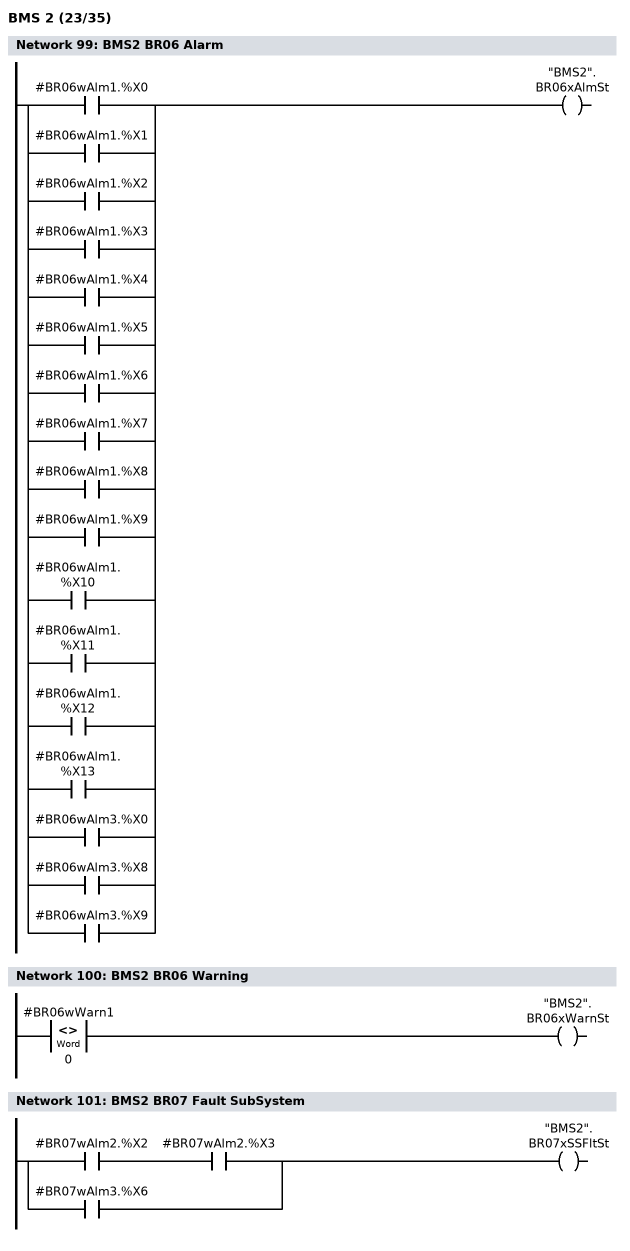
   RUNG wire#powerrail
      Contact( #BR06wAlm1.%X0 )
      wire#w1
      Coil( "BMS2".BR06xAlmSt )
   END_RUNG
   RUNG wire#powerrail
      Contact( #BR06wAlm1.%X1 )
   END_RUNG wire#w1
   RUNG wire#powerrail
      Contact( #BR06wAlm1.%X2 )
   END_RUNG wire#w1
   RUNG wire#powerrail
      Contact( #BR06wAlm1.%X3 )
   END_RUNG wire#w1
   RUNG wire#powerrail
      Contact( #BR06wAlm1.%X4 )
   END_RUNG wire#w1
   RUNG wire#powerrail
      Contact( #BR06wAlm1.%X5 )
   END_RUNG wire#w1
   RUNG wire#powerrail
      Contact( #BR06wAlm1.%X6 )
   END_RUNG wire#w1
   RUNG wire#powerrail
      Contact( #BR06wAlm1.%X7 )
   END_RUNG wire#w1
   RUNG wire#powerrail
      Contact( #BR06wAlm1.%X8 )
   END_RUNG wire#w1
   RUNG wire#powerrail
      Contact( #BR06wAlm1.%X9 )
   END_RUNG wire#w1
   RUNG wire#powerrail
      Contact( #BR06wAlm1.%X10 )
   END_RUNG wire#w1
   RUNG wire#powerrail
      Contact( #BR06wAlm1.%X11 )
   END_RUNG wire#w1
   RUNG wire#powerrail
      Contact( #BR06wAlm1.%X12 )
   END_RUNG wire#w1
   RUNG wire#powerrail
      Contact( #BR06wAlm1.%X13 )
   END_RUNG wire#w1
   RUNG wire#powerrail
      Contact( #BR06wAlm3.%X0 )
   END_RUNG wire#w1
   RUNG wire#powerrail
      Contact( #BR06wAlm3.%X8 )
   END_RUNG wire#w1
   RUNG wire#powerrail
      Contact( #BR06wAlm3.%X9 )
   END_RUNG wire#w1
   // the same network as SCL:
   "BMS2".BR06xAlmSt := #BR06wAlm1.%X0 OR #BR06wAlm1.%X1 OR #BR06wAlm1.%X2 OR #BR06wAlm1.%X3 OR #BR06wAlm1.%X4 OR #BR06wAlm1.%X5 OR #BR06wAlm1.%X6 OR #BR06wAlm1.%X7 OR #BR06wAlm1.%X8 OR #BR06wAlm1.%X9 OR #BR06wAlm1.%X10 OR #BR06wAlm1.%X11 OR #BR06wAlm1.%X12 OR #BR06wAlm1.%X13 OR #BR06wAlm3.%X0 OR #BR06wAlm3.%X8 OR #BR06wAlm3.%X9;
END_REGION

REGION Network 100: BMS2 BR06 Warning
   RUNG wire#powerrail
      { S7_Templates := "SrcType := Word" } NE_Contact(in1 := #BR06wWarn1, in2 := 0)
      Coil( "BMS2".BR06xWarnSt )
   END_RUNG
   // the same network as SCL:
   "BMS2".BR06xWarnSt := #BR06wWarn1 <> 0;
END_REGION

REGION Network 101: BMS2 BR07 Fault SubSystem
   RUNG wire#powerrail
      Contact( #BR07wAlm2.%X2 )
      Contact( #BR07wAlm2.%X3 )
      wire#w1
      Coil( "BMS2".BR07xSSFltSt )
   END_RUNG
   RUNG wire#powerrail
      Contact( #BR07wAlm3.%X6 )
   END_RUNG wire#w1
   // the same network as SCL:
   "BMS2".BR07xSSFltSt := (#BR07wAlm2.%X2 AND #BR07wAlm2.%X3) OR #BR07wAlm3.%X6;
END_REGION

REGION Network 102: BMS2 BR07 Fault
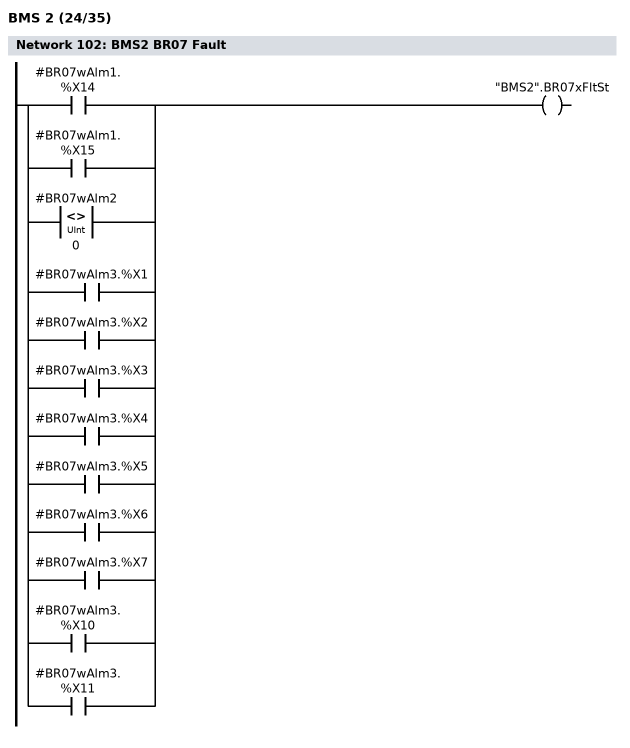
   RUNG wire#powerrail
      Contact( #BR07wAlm1.%X14 )
      wire#w1
      Coil( "BMS2".BR07xFltSt )
   END_RUNG
   RUNG wire#powerrail
      Contact( #BR07wAlm1.%X15 )
   END_RUNG wire#w1
   RUNG wire#powerrail
      { S7_Templates := "SrcType := UInt" } NE_Contact(in1 := #BR07wAlm2, in2 := 0)
   END_RUNG wire#w1
   RUNG wire#powerrail
      Contact( #BR07wAlm3.%X1 )
   END_RUNG wire#w1
   RUNG wire#powerrail
      Contact( #BR07wAlm3.%X2 )
   END_RUNG wire#w1
   RUNG wire#powerrail
      Contact( #BR07wAlm3.%X3 )
   END_RUNG wire#w1
   RUNG wire#powerrail
      Contact( #BR07wAlm3.%X4 )
   END_RUNG wire#w1
   RUNG wire#powerrail
      Contact( #BR07wAlm3.%X5 )
   END_RUNG wire#w1
   RUNG wire#powerrail
      Contact( #BR07wAlm3.%X6 )
   END_RUNG wire#w1
   RUNG wire#powerrail
      Contact( #BR07wAlm3.%X7 )
   END_RUNG wire#w1
   RUNG wire#powerrail
      Contact( #BR07wAlm3.%X10 )
   END_RUNG wire#w1
   RUNG wire#powerrail
      Contact( #BR07wAlm3.%X11 )
   END_RUNG wire#w1
   // the same network as SCL:
   "BMS2".BR07xFltSt := #BR07wAlm1.%X14 OR #BR07wAlm1.%X15 OR (#BR07wAlm2 <> 0) OR #BR07wAlm3.%X1 OR #BR07wAlm3.%X2 OR #BR07wAlm3.%X3 OR #BR07wAlm3.%X4 OR #BR07wAlm3.%X5 OR #BR07wAlm3.%X6 OR #BR07wAlm3.%X7 OR #BR07wAlm3.%X10 OR #BR07wAlm3.%X11;
END_REGION

REGION Network 103: BMS2 BR07 Alarm
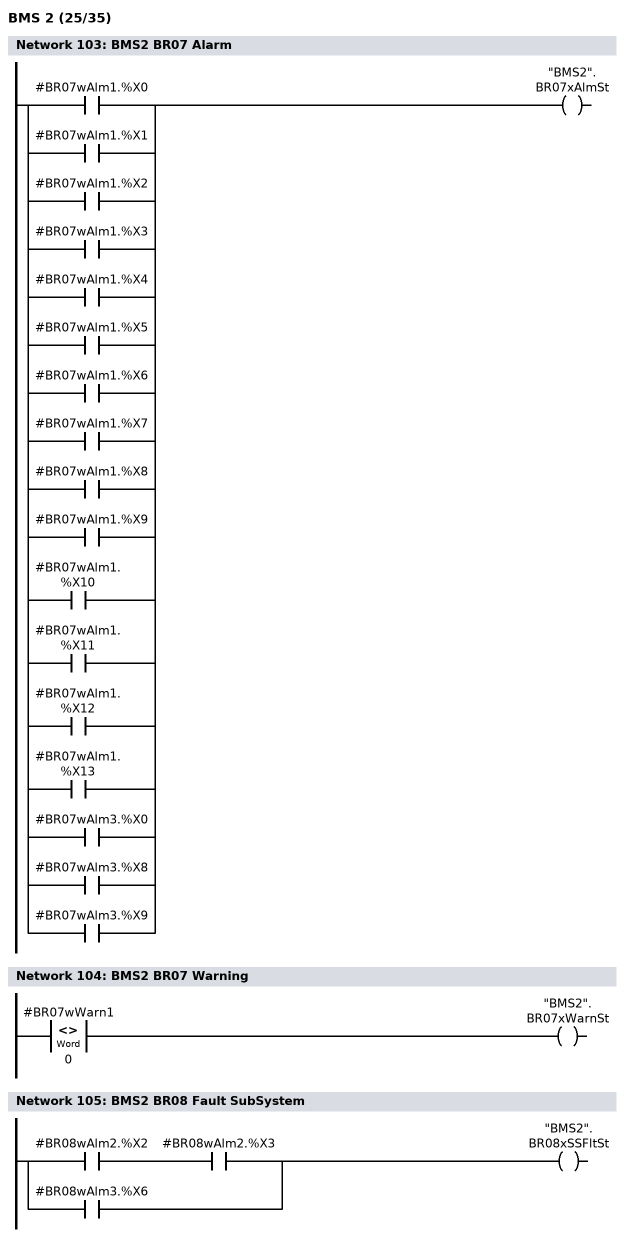
   RUNG wire#powerrail
      Contact( #BR07wAlm1.%X0 )
      wire#w1
      Coil( "BMS2".BR07xAlmSt )
   END_RUNG
   RUNG wire#powerrail
      Contact( #BR07wAlm1.%X1 )
   END_RUNG wire#w1
   RUNG wire#powerrail
      Contact( #BR07wAlm1.%X2 )
   END_RUNG wire#w1
   RUNG wire#powerrail
      Contact( #BR07wAlm1.%X3 )
   END_RUNG wire#w1
   RUNG wire#powerrail
      Contact( #BR07wAlm1.%X4 )
   END_RUNG wire#w1
   RUNG wire#powerrail
      Contact( #BR07wAlm1.%X5 )
   END_RUNG wire#w1
   RUNG wire#powerrail
      Contact( #BR07wAlm1.%X6 )
   END_RUNG wire#w1
   RUNG wire#powerrail
      Contact( #BR07wAlm1.%X7 )
   END_RUNG wire#w1
   RUNG wire#powerrail
      Contact( #BR07wAlm1.%X8 )
   END_RUNG wire#w1
   RUNG wire#powerrail
      Contact( #BR07wAlm1.%X9 )
   END_RUNG wire#w1
   RUNG wire#powerrail
      Contact( #BR07wAlm1.%X10 )
   END_RUNG wire#w1
   RUNG wire#powerrail
      Contact( #BR07wAlm1.%X11 )
   END_RUNG wire#w1
   RUNG wire#powerrail
      Contact( #BR07wAlm1.%X12 )
   END_RUNG wire#w1
   RUNG wire#powerrail
      Contact( #BR07wAlm1.%X13 )
   END_RUNG wire#w1
   RUNG wire#powerrail
      Contact( #BR07wAlm3.%X0 )
   END_RUNG wire#w1
   RUNG wire#powerrail
      Contact( #BR07wAlm3.%X8 )
   END_RUNG wire#w1
   RUNG wire#powerrail
      Contact( #BR07wAlm3.%X9 )
   END_RUNG wire#w1
   // the same network as SCL:
   "BMS2".BR07xAlmSt := #BR07wAlm1.%X0 OR #BR07wAlm1.%X1 OR #BR07wAlm1.%X2 OR #BR07wAlm1.%X3 OR #BR07wAlm1.%X4 OR #BR07wAlm1.%X5 OR #BR07wAlm1.%X6 OR #BR07wAlm1.%X7 OR #BR07wAlm1.%X8 OR #BR07wAlm1.%X9 OR #BR07wAlm1.%X10 OR #BR07wAlm1.%X11 OR #BR07wAlm1.%X12 OR #BR07wAlm1.%X13 OR #BR07wAlm3.%X0 OR #BR07wAlm3.%X8 OR #BR07wAlm3.%X9;
END_REGION

REGION Network 104: BMS2 BR07 Warning
   RUNG wire#powerrail
      { S7_Templates := "SrcType := Word" } NE_Contact(in1 := #BR07wWarn1, in2 := 0)
      Coil( "BMS2".BR07xWarnSt )
   END_RUNG
   // the same network as SCL:
   "BMS2".BR07xWarnSt := #BR07wWarn1 <> 0;
END_REGION

REGION Network 105: BMS2 BR08 Fault SubSystem
   RUNG wire#powerrail
      Contact( #BR08wAlm2.%X2 )
      Contact( #BR08wAlm2.%X3 )
      wire#w1
      Coil( "BMS2".BR08xSSFltSt )
   END_RUNG
   RUNG wire#powerrail
      Contact( #BR08wAlm3.%X6 )
   END_RUNG wire#w1
   // the same network as SCL:
   "BMS2".BR08xSSFltSt := (#BR08wAlm2.%X2 AND #BR08wAlm2.%X3) OR #BR08wAlm3.%X6;
END_REGION

REGION Network 106: BMS2 BR08 Fault
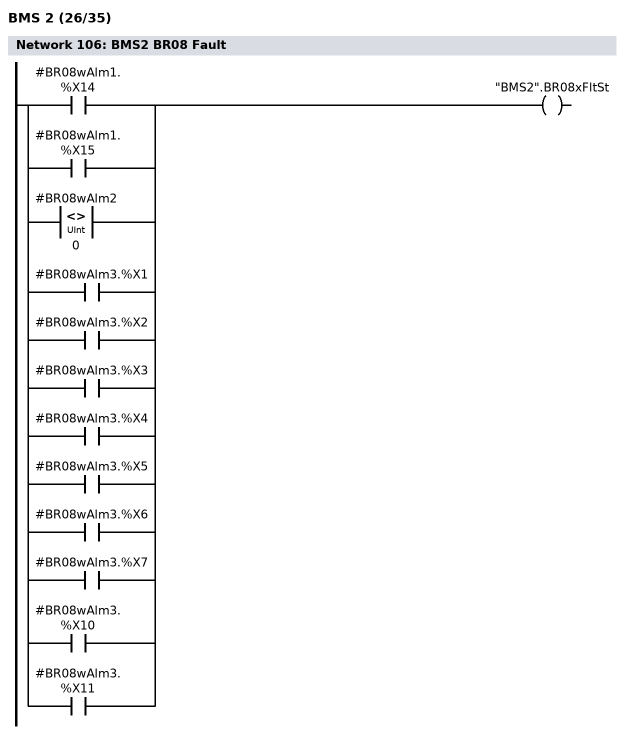
   RUNG wire#powerrail
      Contact( #BR08wAlm1.%X14 )
      wire#w1
      Coil( "BMS2".BR08xFltSt )
   END_RUNG
   RUNG wire#powerrail
      Contact( #BR08wAlm1.%X15 )
   END_RUNG wire#w1
   RUNG wire#powerrail
      { S7_Templates := "SrcType := UInt" } NE_Contact(in1 := #BR08wAlm2, in2 := 0)
   END_RUNG wire#w1
   RUNG wire#powerrail
      Contact( #BR08wAlm3.%X1 )
   END_RUNG wire#w1
   RUNG wire#powerrail
      Contact( #BR08wAlm3.%X2 )
   END_RUNG wire#w1
   RUNG wire#powerrail
      Contact( #BR08wAlm3.%X3 )
   END_RUNG wire#w1
   RUNG wire#powerrail
      Contact( #BR08wAlm3.%X4 )
   END_RUNG wire#w1
   RUNG wire#powerrail
      Contact( #BR08wAlm3.%X5 )
   END_RUNG wire#w1
   RUNG wire#powerrail
      Contact( #BR08wAlm3.%X6 )
   END_RUNG wire#w1
   RUNG wire#powerrail
      Contact( #BR08wAlm3.%X7 )
   END_RUNG wire#w1
   RUNG wire#powerrail
      Contact( #BR08wAlm3.%X10 )
   END_RUNG wire#w1
   RUNG wire#powerrail
      Contact( #BR08wAlm3.%X11 )
   END_RUNG wire#w1
   // the same network as SCL:
   "BMS2".BR08xFltSt := #BR08wAlm1.%X14 OR #BR08wAlm1.%X15 OR (#BR08wAlm2 <> 0) OR #BR08wAlm3.%X1 OR #BR08wAlm3.%X2 OR #BR08wAlm3.%X3 OR #BR08wAlm3.%X4 OR #BR08wAlm3.%X5 OR #BR08wAlm3.%X6 OR #BR08wAlm3.%X7 OR #BR08wAlm3.%X10 OR #BR08wAlm3.%X11;
END_REGION

REGION Network 107: BMS2 BR08 Alarm
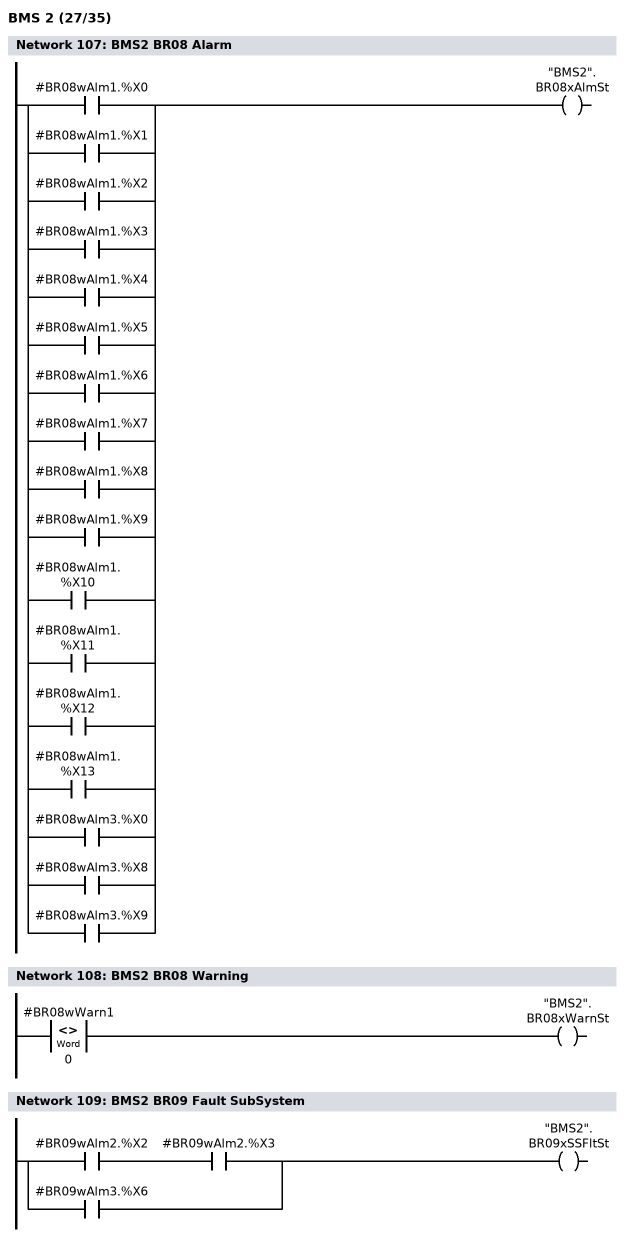
   RUNG wire#powerrail
      Contact( #BR08wAlm1.%X0 )
      wire#w1
      Coil( "BMS2".BR08xAlmSt )
   END_RUNG
   RUNG wire#powerrail
      Contact( #BR08wAlm1.%X1 )
   END_RUNG wire#w1
   RUNG wire#powerrail
      Contact( #BR08wAlm1.%X2 )
   END_RUNG wire#w1
   RUNG wire#powerrail
      Contact( #BR08wAlm1.%X3 )
   END_RUNG wire#w1
   RUNG wire#powerrail
      Contact( #BR08wAlm1.%X4 )
   END_RUNG wire#w1
   RUNG wire#powerrail
      Contact( #BR08wAlm1.%X5 )
   END_RUNG wire#w1
   RUNG wire#powerrail
      Contact( #BR08wAlm1.%X6 )
   END_RUNG wire#w1
   RUNG wire#powerrail
      Contact( #BR08wAlm1.%X7 )
   END_RUNG wire#w1
   RUNG wire#powerrail
      Contact( #BR08wAlm1.%X8 )
   END_RUNG wire#w1
   RUNG wire#powerrail
      Contact( #BR08wAlm1.%X9 )
   END_RUNG wire#w1
   RUNG wire#powerrail
      Contact( #BR08wAlm1.%X10 )
   END_RUNG wire#w1
   RUNG wire#powerrail
      Contact( #BR08wAlm1.%X11 )
   END_RUNG wire#w1
   RUNG wire#powerrail
      Contact( #BR08wAlm1.%X12 )
   END_RUNG wire#w1
   RUNG wire#powerrail
      Contact( #BR08wAlm1.%X13 )
   END_RUNG wire#w1
   RUNG wire#powerrail
      Contact( #BR08wAlm3.%X0 )
   END_RUNG wire#w1
   RUNG wire#powerrail
      Contact( #BR08wAlm3.%X8 )
   END_RUNG wire#w1
   RUNG wire#powerrail
      Contact( #BR08wAlm3.%X9 )
   END_RUNG wire#w1
   // the same network as SCL:
   "BMS2".BR08xAlmSt := #BR08wAlm1.%X0 OR #BR08wAlm1.%X1 OR #BR08wAlm1.%X2 OR #BR08wAlm1.%X3 OR #BR08wAlm1.%X4 OR #BR08wAlm1.%X5 OR #BR08wAlm1.%X6 OR #BR08wAlm1.%X7 OR #BR08wAlm1.%X8 OR #BR08wAlm1.%X9 OR #BR08wAlm1.%X10 OR #BR08wAlm1.%X11 OR #BR08wAlm1.%X12 OR #BR08wAlm1.%X13 OR #BR08wAlm3.%X0 OR #BR08wAlm3.%X8 OR #BR08wAlm3.%X9;
END_REGION

REGION Network 108: BMS2 BR08 Warning
   RUNG wire#powerrail
      { S7_Templates := "SrcType := Word" } NE_Contact(in1 := #BR08wWarn1, in2 := 0)
      Coil( "BMS2".BR08xWarnSt )
   END_RUNG
   // the same network as SCL:
   "BMS2".BR08xWarnSt := #BR08wWarn1 <> 0;
END_REGION

REGION Network 109: BMS2 BR09 Fault SubSystem
   RUNG wire#powerrail
      Contact( #BR09wAlm2.%X2 )
      Contact( #BR09wAlm2.%X3 )
      wire#w1
      Coil( "BMS2".BR09xSSFltSt )
   END_RUNG
   RUNG wire#powerrail
      Contact( #BR09wAlm3.%X6 )
   END_RUNG wire#w1
   // the same network as SCL:
   "BMS2".BR09xSSFltSt := (#BR09wAlm2.%X2 AND #BR09wAlm2.%X3) OR #BR09wAlm3.%X6;
END_REGION

REGION Network 110: BMS2 BR09 Fault
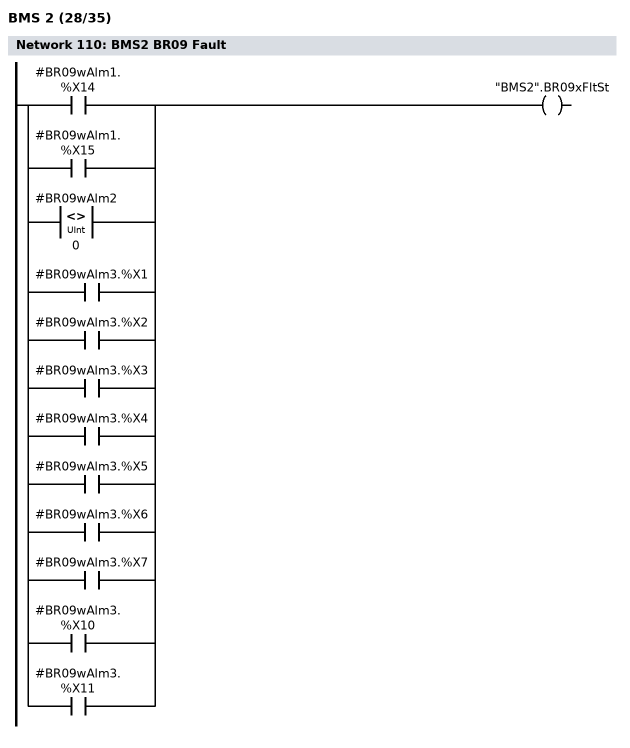
   RUNG wire#powerrail
      Contact( #BR09wAlm1.%X14 )
      wire#w1
      Coil( "BMS2".BR09xFltSt )
   END_RUNG
   RUNG wire#powerrail
      Contact( #BR09wAlm1.%X15 )
   END_RUNG wire#w1
   RUNG wire#powerrail
      { S7_Templates := "SrcType := UInt" } NE_Contact(in1 := #BR09wAlm2, in2 := 0)
   END_RUNG wire#w1
   RUNG wire#powerrail
      Contact( #BR09wAlm3.%X1 )
   END_RUNG wire#w1
   RUNG wire#powerrail
      Contact( #BR09wAlm3.%X2 )
   END_RUNG wire#w1
   RUNG wire#powerrail
      Contact( #BR09wAlm3.%X3 )
   END_RUNG wire#w1
   RUNG wire#powerrail
      Contact( #BR09wAlm3.%X4 )
   END_RUNG wire#w1
   RUNG wire#powerrail
      Contact( #BR09wAlm3.%X5 )
   END_RUNG wire#w1
   RUNG wire#powerrail
      Contact( #BR09wAlm3.%X6 )
   END_RUNG wire#w1
   RUNG wire#powerrail
      Contact( #BR09wAlm3.%X7 )
   END_RUNG wire#w1
   RUNG wire#powerrail
      Contact( #BR09wAlm3.%X10 )
   END_RUNG wire#w1
   RUNG wire#powerrail
      Contact( #BR09wAlm3.%X11 )
   END_RUNG wire#w1
   // the same network as SCL:
   "BMS2".BR09xFltSt := #BR09wAlm1.%X14 OR #BR09wAlm1.%X15 OR (#BR09wAlm2 <> 0) OR #BR09wAlm3.%X1 OR #BR09wAlm3.%X2 OR #BR09wAlm3.%X3 OR #BR09wAlm3.%X4 OR #BR09wAlm3.%X5 OR #BR09wAlm3.%X6 OR #BR09wAlm3.%X7 OR #BR09wAlm3.%X10 OR #BR09wAlm3.%X11;
END_REGION

REGION Network 111: BMS2 BR09 Alarm
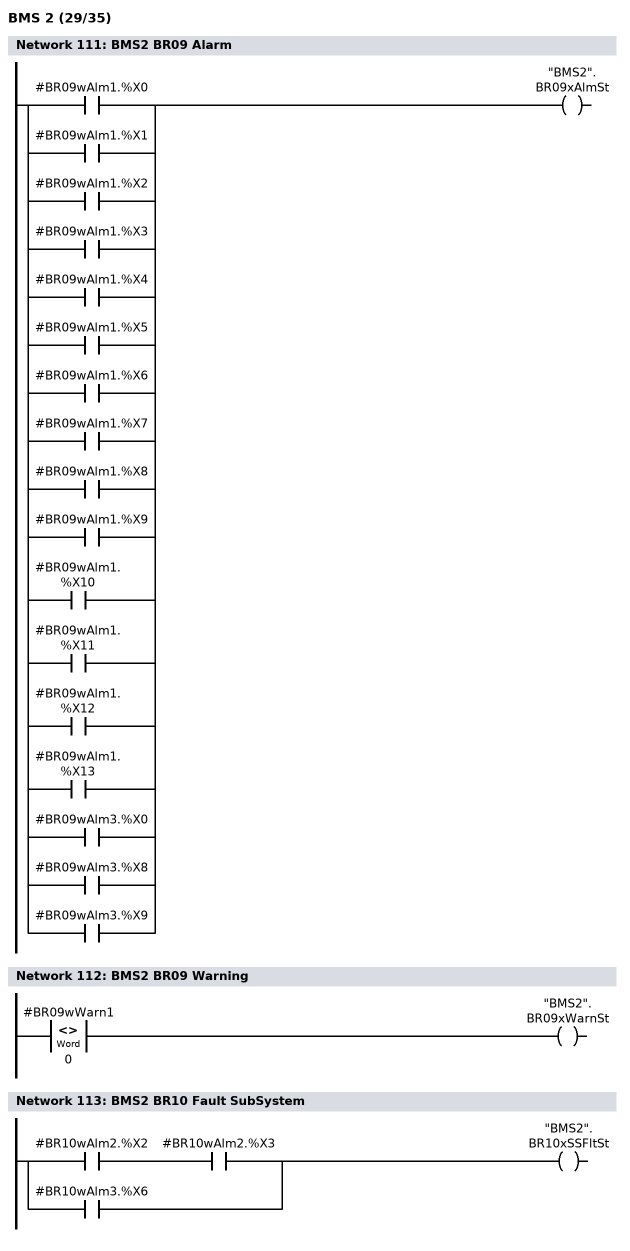
   RUNG wire#powerrail
      Contact( #BR09wAlm1.%X0 )
      wire#w1
      Coil( "BMS2".BR09xAlmSt )
   END_RUNG
   RUNG wire#powerrail
      Contact( #BR09wAlm1.%X1 )
   END_RUNG wire#w1
   RUNG wire#powerrail
      Contact( #BR09wAlm1.%X2 )
   END_RUNG wire#w1
   RUNG wire#powerrail
      Contact( #BR09wAlm1.%X3 )
   END_RUNG wire#w1
   RUNG wire#powerrail
      Contact( #BR09wAlm1.%X4 )
   END_RUNG wire#w1
   RUNG wire#powerrail
      Contact( #BR09wAlm1.%X5 )
   END_RUNG wire#w1
   RUNG wire#powerrail
      Contact( #BR09wAlm1.%X6 )
   END_RUNG wire#w1
   RUNG wire#powerrail
      Contact( #BR09wAlm1.%X7 )
   END_RUNG wire#w1
   RUNG wire#powerrail
      Contact( #BR09wAlm1.%X8 )
   END_RUNG wire#w1
   RUNG wire#powerrail
      Contact( #BR09wAlm1.%X9 )
   END_RUNG wire#w1
   RUNG wire#powerrail
      Contact( #BR09wAlm1.%X10 )
   END_RUNG wire#w1
   RUNG wire#powerrail
      Contact( #BR09wAlm1.%X11 )
   END_RUNG wire#w1
   RUNG wire#powerrail
      Contact( #BR09wAlm1.%X12 )
   END_RUNG wire#w1
   RUNG wire#powerrail
      Contact( #BR09wAlm1.%X13 )
   END_RUNG wire#w1
   RUNG wire#powerrail
      Contact( #BR09wAlm3.%X0 )
   END_RUNG wire#w1
   RUNG wire#powerrail
      Contact( #BR09wAlm3.%X8 )
   END_RUNG wire#w1
   RUNG wire#powerrail
      Contact( #BR09wAlm3.%X9 )
   END_RUNG wire#w1
   // the same network as SCL:
   "BMS2".BR09xAlmSt := #BR09wAlm1.%X0 OR #BR09wAlm1.%X1 OR #BR09wAlm1.%X2 OR #BR09wAlm1.%X3 OR #BR09wAlm1.%X4 OR #BR09wAlm1.%X5 OR #BR09wAlm1.%X6 OR #BR09wAlm1.%X7 OR #BR09wAlm1.%X8 OR #BR09wAlm1.%X9 OR #BR09wAlm1.%X10 OR #BR09wAlm1.%X11 OR #BR09wAlm1.%X12 OR #BR09wAlm1.%X13 OR #BR09wAlm3.%X0 OR #BR09wAlm3.%X8 OR #BR09wAlm3.%X9;
END_REGION

REGION Network 112: BMS2 BR09 Warning
   RUNG wire#powerrail
      { S7_Templates := "SrcType := Word" } NE_Contact(in1 := #BR09wWarn1, in2 := 0)
      Coil( "BMS2".BR09xWarnSt )
   END_RUNG
   // the same network as SCL:
   "BMS2".BR09xWarnSt := #BR09wWarn1 <> 0;
END_REGION

REGION Network 113: BMS2 BR10 Fault SubSystem
   RUNG wire#powerrail
      Contact( #BR10wAlm2.%X2 )
      Contact( #BR10wAlm2.%X3 )
      wire#w1
      Coil( "BMS2".BR10xSSFltSt )
   END_RUNG
   RUNG wire#powerrail
      Contact( #BR10wAlm3.%X6 )
   END_RUNG wire#w1
   // the same network as SCL:
   "BMS2".BR10xSSFltSt := (#BR10wAlm2.%X2 AND #BR10wAlm2.%X3) OR #BR10wAlm3.%X6;
END_REGION

REGION Network 114: BMS2 BR10 Fault
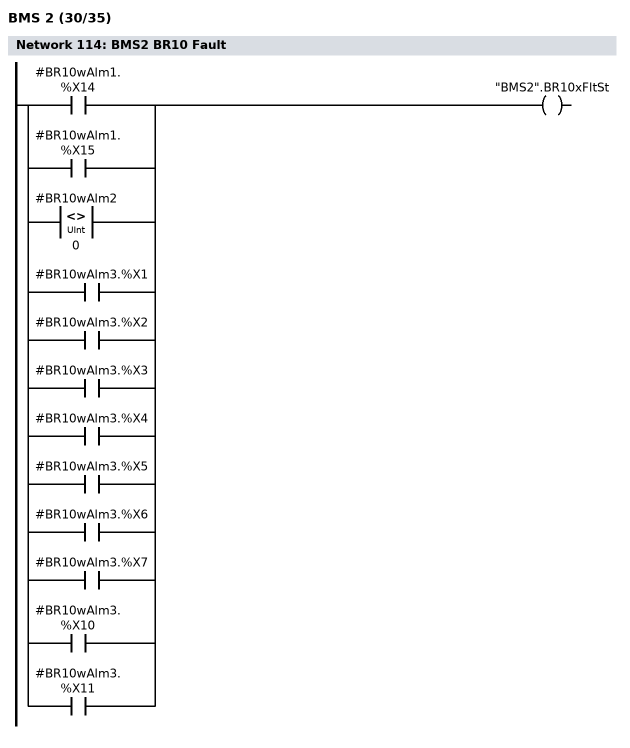
   RUNG wire#powerrail
      Contact( #BR10wAlm1.%X14 )
      wire#w1
      Coil( "BMS2".BR10xFltSt )
   END_RUNG
   RUNG wire#powerrail
      Contact( #BR10wAlm1.%X15 )
   END_RUNG wire#w1
   RUNG wire#powerrail
      { S7_Templates := "SrcType := UInt" } NE_Contact(in1 := #BR10wAlm2, in2 := 0)
   END_RUNG wire#w1
   RUNG wire#powerrail
      Contact( #BR10wAlm3.%X1 )
   END_RUNG wire#w1
   RUNG wire#powerrail
      Contact( #BR10wAlm3.%X2 )
   END_RUNG wire#w1
   RUNG wire#powerrail
      Contact( #BR10wAlm3.%X3 )
   END_RUNG wire#w1
   RUNG wire#powerrail
      Contact( #BR10wAlm3.%X4 )
   END_RUNG wire#w1
   RUNG wire#powerrail
      Contact( #BR10wAlm3.%X5 )
   END_RUNG wire#w1
   RUNG wire#powerrail
      Contact( #BR10wAlm3.%X6 )
   END_RUNG wire#w1
   RUNG wire#powerrail
      Contact( #BR10wAlm3.%X7 )
   END_RUNG wire#w1
   RUNG wire#powerrail
      Contact( #BR10wAlm3.%X10 )
   END_RUNG wire#w1
   RUNG wire#powerrail
      Contact( #BR10wAlm3.%X11 )
   END_RUNG wire#w1
   // the same network as SCL:
   "BMS2".BR10xFltSt := #BR10wAlm1.%X14 OR #BR10wAlm1.%X15 OR (#BR10wAlm2 <> 0) OR #BR10wAlm3.%X1 OR #BR10wAlm3.%X2 OR #BR10wAlm3.%X3 OR #BR10wAlm3.%X4 OR #BR10wAlm3.%X5 OR #BR10wAlm3.%X6 OR #BR10wAlm3.%X7 OR #BR10wAlm3.%X10 OR #BR10wAlm3.%X11;
END_REGION

REGION Network 115: BMS2 BR10 Alarm
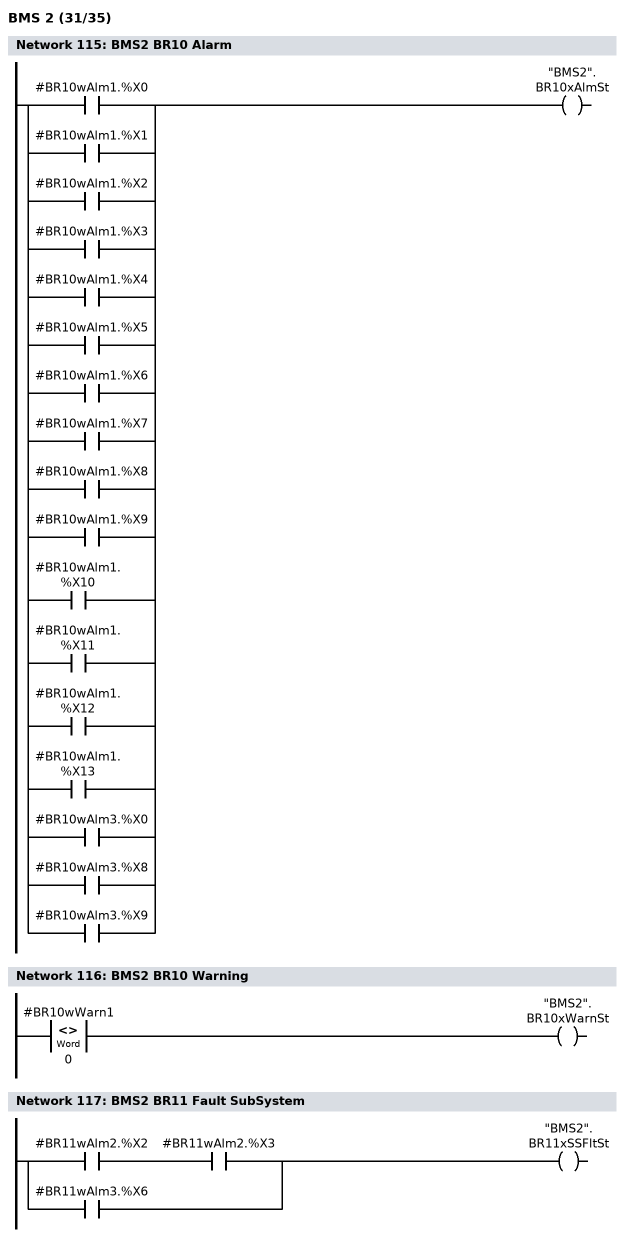
   RUNG wire#powerrail
      Contact( #BR10wAlm1.%X0 )
      wire#w1
      Coil( "BMS2".BR10xAlmSt )
   END_RUNG
   RUNG wire#powerrail
      Contact( #BR10wAlm1.%X1 )
   END_RUNG wire#w1
   RUNG wire#powerrail
      Contact( #BR10wAlm1.%X2 )
   END_RUNG wire#w1
   RUNG wire#powerrail
      Contact( #BR10wAlm1.%X3 )
   END_RUNG wire#w1
   RUNG wire#powerrail
      Contact( #BR10wAlm1.%X4 )
   END_RUNG wire#w1
   RUNG wire#powerrail
      Contact( #BR10wAlm1.%X5 )
   END_RUNG wire#w1
   RUNG wire#powerrail
      Contact( #BR10wAlm1.%X6 )
   END_RUNG wire#w1
   RUNG wire#powerrail
      Contact( #BR10wAlm1.%X7 )
   END_RUNG wire#w1
   RUNG wire#powerrail
      Contact( #BR10wAlm1.%X8 )
   END_RUNG wire#w1
   RUNG wire#powerrail
      Contact( #BR10wAlm1.%X9 )
   END_RUNG wire#w1
   RUNG wire#powerrail
      Contact( #BR10wAlm1.%X10 )
   END_RUNG wire#w1
   RUNG wire#powerrail
      Contact( #BR10wAlm1.%X11 )
   END_RUNG wire#w1
   RUNG wire#powerrail
      Contact( #BR10wAlm1.%X12 )
   END_RUNG wire#w1
   RUNG wire#powerrail
      Contact( #BR10wAlm1.%X13 )
   END_RUNG wire#w1
   RUNG wire#powerrail
      Contact( #BR10wAlm3.%X0 )
   END_RUNG wire#w1
   RUNG wire#powerrail
      Contact( #BR10wAlm3.%X8 )
   END_RUNG wire#w1
   RUNG wire#powerrail
      Contact( #BR10wAlm3.%X9 )
   END_RUNG wire#w1
   // the same network as SCL:
   "BMS2".BR10xAlmSt := #BR10wAlm1.%X0 OR #BR10wAlm1.%X1 OR #BR10wAlm1.%X2 OR #BR10wAlm1.%X3 OR #BR10wAlm1.%X4 OR #BR10wAlm1.%X5 OR #BR10wAlm1.%X6 OR #BR10wAlm1.%X7 OR #BR10wAlm1.%X8 OR #BR10wAlm1.%X9 OR #BR10wAlm1.%X10 OR #BR10wAlm1.%X11 OR #BR10wAlm1.%X12 OR #BR10wAlm1.%X13 OR #BR10wAlm3.%X0 OR #BR10wAlm3.%X8 OR #BR10wAlm3.%X9;
END_REGION

REGION Network 116: BMS2 BR10 Warning
   RUNG wire#powerrail
      { S7_Templates := "SrcType := Word" } NE_Contact(in1 := #BR10wWarn1, in2 := 0)
      Coil( "BMS2".BR10xWarnSt )
   END_RUNG
   // the same network as SCL:
   "BMS2".BR10xWarnSt := #BR10wWarn1 <> 0;
END_REGION

REGION Network 117: BMS2 BR11 Fault SubSystem
   RUNG wire#powerrail
      Contact( #BR11wAlm2.%X2 )
      Contact( #BR11wAlm2.%X3 )
      wire#w1
      Coil( "BMS2".BR11xSSFltSt )
   END_RUNG
   RUNG wire#powerrail
      Contact( #BR11wAlm3.%X6 )
   END_RUNG wire#w1
   // the same network as SCL:
   "BMS2".BR11xSSFltSt := (#BR11wAlm2.%X2 AND #BR11wAlm2.%X3) OR #BR11wAlm3.%X6;
END_REGION

REGION Network 118: BMS2 BR11 Fault
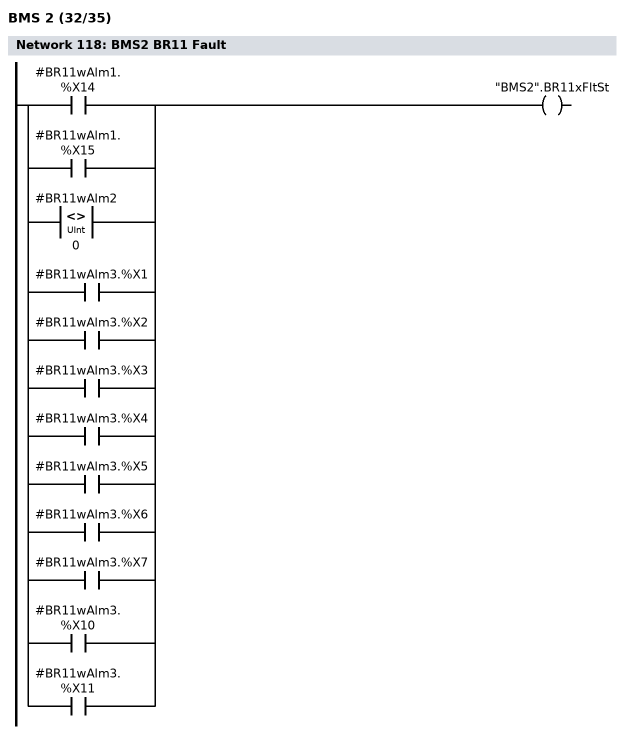
   RUNG wire#powerrail
      Contact( #BR11wAlm1.%X14 )
      wire#w1
      Coil( "BMS2".BR11xFltSt )
   END_RUNG
   RUNG wire#powerrail
      Contact( #BR11wAlm1.%X15 )
   END_RUNG wire#w1
   RUNG wire#powerrail
      { S7_Templates := "SrcType := UInt" } NE_Contact(in1 := #BR11wAlm2, in2 := 0)
   END_RUNG wire#w1
   RUNG wire#powerrail
      Contact( #BR11wAlm3.%X1 )
   END_RUNG wire#w1
   RUNG wire#powerrail
      Contact( #BR11wAlm3.%X2 )
   END_RUNG wire#w1
   RUNG wire#powerrail
      Contact( #BR11wAlm3.%X3 )
   END_RUNG wire#w1
   RUNG wire#powerrail
      Contact( #BR11wAlm3.%X4 )
   END_RUNG wire#w1
   RUNG wire#powerrail
      Contact( #BR11wAlm3.%X5 )
   END_RUNG wire#w1
   RUNG wire#powerrail
      Contact( #BR11wAlm3.%X6 )
   END_RUNG wire#w1
   RUNG wire#powerrail
      Contact( #BR11wAlm3.%X7 )
   END_RUNG wire#w1
   RUNG wire#powerrail
      Contact( #BR11wAlm3.%X10 )
   END_RUNG wire#w1
   RUNG wire#powerrail
      Contact( #BR11wAlm3.%X11 )
   END_RUNG wire#w1
   // the same network as SCL:
   "BMS2".BR11xFltSt := #BR11wAlm1.%X14 OR #BR11wAlm1.%X15 OR (#BR11wAlm2 <> 0) OR #BR11wAlm3.%X1 OR #BR11wAlm3.%X2 OR #BR11wAlm3.%X3 OR #BR11wAlm3.%X4 OR #BR11wAlm3.%X5 OR #BR11wAlm3.%X6 OR #BR11wAlm3.%X7 OR #BR11wAlm3.%X10 OR #BR11wAlm3.%X11;
END_REGION

REGION Network 119: BMS2 BR11 Alarm
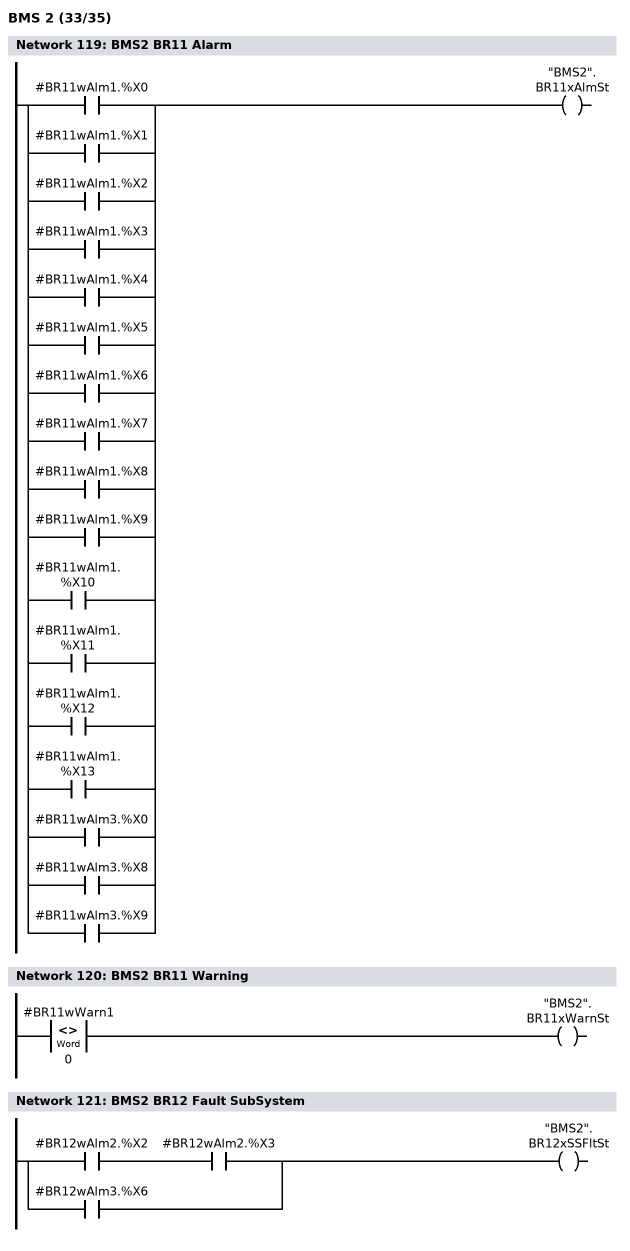
   RUNG wire#powerrail
      Contact( #BR11wAlm1.%X0 )
      wire#w1
      Coil( "BMS2".BR11xAlmSt )
   END_RUNG
   RUNG wire#powerrail
      Contact( #BR11wAlm1.%X1 )
   END_RUNG wire#w1
   RUNG wire#powerrail
      Contact( #BR11wAlm1.%X2 )
   END_RUNG wire#w1
   RUNG wire#powerrail
      Contact( #BR11wAlm1.%X3 )
   END_RUNG wire#w1
   RUNG wire#powerrail
      Contact( #BR11wAlm1.%X4 )
   END_RUNG wire#w1
   RUNG wire#powerrail
      Contact( #BR11wAlm1.%X5 )
   END_RUNG wire#w1
   RUNG wire#powerrail
      Contact( #BR11wAlm1.%X6 )
   END_RUNG wire#w1
   RUNG wire#powerrail
      Contact( #BR11wAlm1.%X7 )
   END_RUNG wire#w1
   RUNG wire#powerrail
      Contact( #BR11wAlm1.%X8 )
   END_RUNG wire#w1
   RUNG wire#powerrail
      Contact( #BR11wAlm1.%X9 )
   END_RUNG wire#w1
   RUNG wire#powerrail
      Contact( #BR11wAlm1.%X10 )
   END_RUNG wire#w1
   RUNG wire#powerrail
      Contact( #BR11wAlm1.%X11 )
   END_RUNG wire#w1
   RUNG wire#powerrail
      Contact( #BR11wAlm1.%X12 )
   END_RUNG wire#w1
   RUNG wire#powerrail
      Contact( #BR11wAlm1.%X13 )
   END_RUNG wire#w1
   RUNG wire#powerrail
      Contact( #BR11wAlm3.%X0 )
   END_RUNG wire#w1
   RUNG wire#powerrail
      Contact( #BR11wAlm3.%X8 )
   END_RUNG wire#w1
   RUNG wire#powerrail
      Contact( #BR11wAlm3.%X9 )
   END_RUNG wire#w1
   // the same network as SCL:
   "BMS2".BR11xAlmSt := #BR11wAlm1.%X0 OR #BR11wAlm1.%X1 OR #BR11wAlm1.%X2 OR #BR11wAlm1.%X3 OR #BR11wAlm1.%X4 OR #BR11wAlm1.%X5 OR #BR11wAlm1.%X6 OR #BR11wAlm1.%X7 OR #BR11wAlm1.%X8 OR #BR11wAlm1.%X9 OR #BR11wAlm1.%X10 OR #BR11wAlm1.%X11 OR #BR11wAlm1.%X12 OR #BR11wAlm1.%X13 OR #BR11wAlm3.%X0 OR #BR11wAlm3.%X8 OR #BR11wAlm3.%X9;
END_REGION

REGION Network 120: BMS2 BR11 Warning
   RUNG wire#powerrail
      { S7_Templates := "SrcType := Word" } NE_Contact(in1 := #BR11wWarn1, in2 := 0)
      Coil( "BMS2".BR11xWarnSt )
   END_RUNG
   // the same network as SCL:
   "BMS2".BR11xWarnSt := #BR11wWarn1 <> 0;
END_REGION

REGION Network 121: BMS2 BR12 Fault SubSystem
   RUNG wire#powerrail
      Contact( #BR12wAlm2.%X2 )
      Contact( #BR12wAlm2.%X3 )
      wire#w1
      Coil( "BMS2".BR12xSSFltSt )
   END_RUNG
   RUNG wire#powerrail
      Contact( #BR12wAlm3.%X6 )
   END_RUNG wire#w1
   // the same network as SCL:
   "BMS2".BR12xSSFltSt := (#BR12wAlm2.%X2 AND #BR12wAlm2.%X3) OR #BR12wAlm3.%X6;
END_REGION

REGION Network 122: BMS2 BR12 Fault
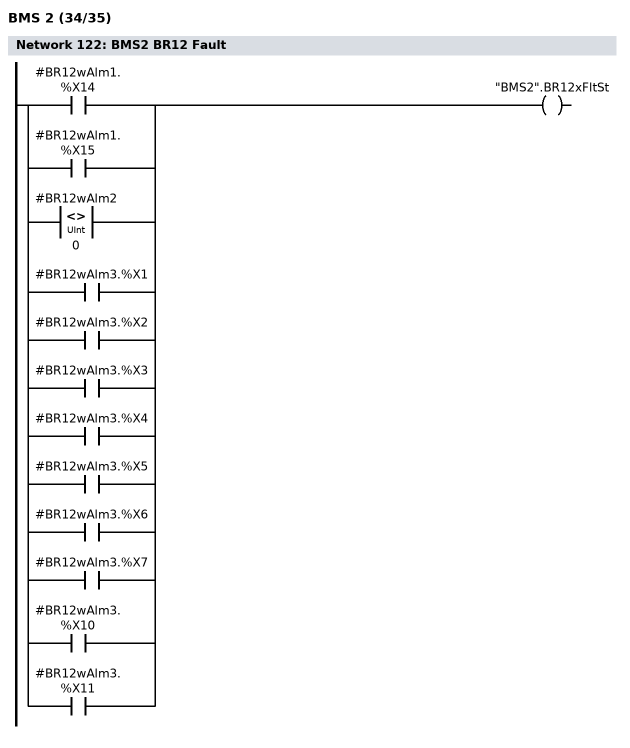
   RUNG wire#powerrail
      Contact( #BR12wAlm1.%X14 )
      wire#w1
      Coil( "BMS2".BR12xFltSt )
   END_RUNG
   RUNG wire#powerrail
      Contact( #BR12wAlm1.%X15 )
   END_RUNG wire#w1
   RUNG wire#powerrail
      { S7_Templates := "SrcType := UInt" } NE_Contact(in1 := #BR12wAlm2, in2 := 0)
   END_RUNG wire#w1
   RUNG wire#powerrail
      Contact( #BR12wAlm3.%X1 )
   END_RUNG wire#w1
   RUNG wire#powerrail
      Contact( #BR12wAlm3.%X2 )
   END_RUNG wire#w1
   RUNG wire#powerrail
      Contact( #BR12wAlm3.%X3 )
   END_RUNG wire#w1
   RUNG wire#powerrail
      Contact( #BR12wAlm3.%X4 )
   END_RUNG wire#w1
   RUNG wire#powerrail
      Contact( #BR12wAlm3.%X5 )
   END_RUNG wire#w1
   RUNG wire#powerrail
      Contact( #BR12wAlm3.%X6 )
   END_RUNG wire#w1
   RUNG wire#powerrail
      Contact( #BR12wAlm3.%X7 )
   END_RUNG wire#w1
   RUNG wire#powerrail
      Contact( #BR12wAlm3.%X10 )
   END_RUNG wire#w1
   RUNG wire#powerrail
      Contact( #BR12wAlm3.%X11 )
   END_RUNG wire#w1
   // the same network as SCL:
   "BMS2".BR12xFltSt := #BR12wAlm1.%X14 OR #BR12wAlm1.%X15 OR (#BR12wAlm2 <> 0) OR #BR12wAlm3.%X1 OR #BR12wAlm3.%X2 OR #BR12wAlm3.%X3 OR #BR12wAlm3.%X4 OR #BR12wAlm3.%X5 OR #BR12wAlm3.%X6 OR #BR12wAlm3.%X7 OR #BR12wAlm3.%X10 OR #BR12wAlm3.%X11;
END_REGION

REGION Network 123: BMS2 BR12 Alarm
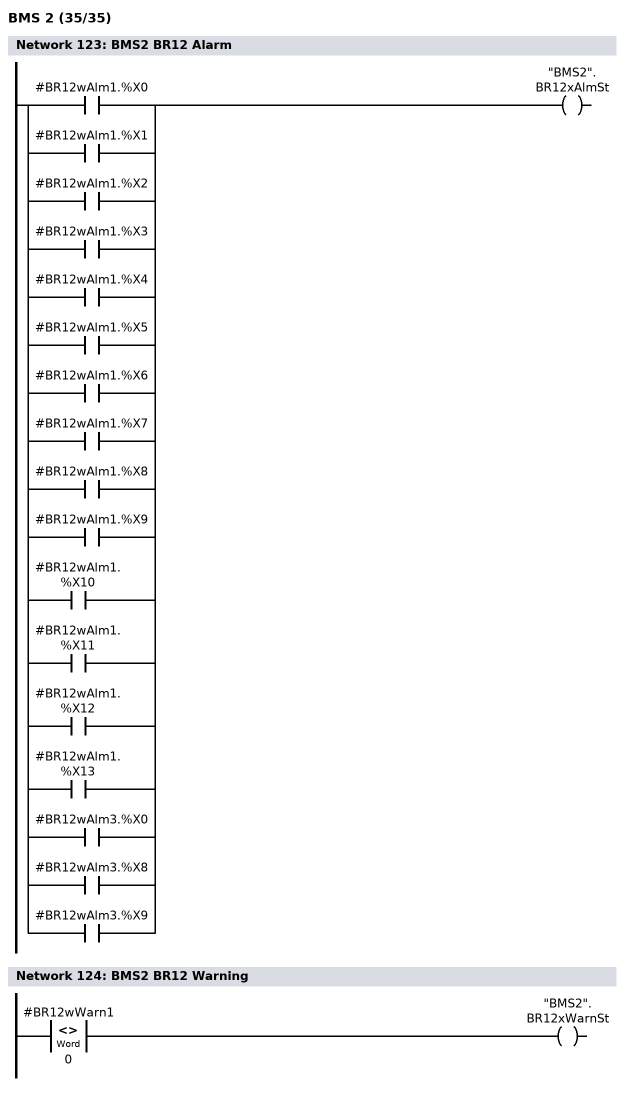
   RUNG wire#powerrail
      Contact( #BR12wAlm1.%X0 )
      wire#w1
      Coil( "BMS2".BR12xAlmSt )
   END_RUNG
   RUNG wire#powerrail
      Contact( #BR12wAlm1.%X1 )
   END_RUNG wire#w1
   RUNG wire#powerrail
      Contact( #BR12wAlm1.%X2 )
   END_RUNG wire#w1
   RUNG wire#powerrail
      Contact( #BR12wAlm1.%X3 )
   END_RUNG wire#w1
   RUNG wire#powerrail
      Contact( #BR12wAlm1.%X4 )
   END_RUNG wire#w1
   RUNG wire#powerrail
      Contact( #BR12wAlm1.%X5 )
   END_RUNG wire#w1
   RUNG wire#powerrail
      Contact( #BR12wAlm1.%X6 )
   END_RUNG wire#w1
   RUNG wire#powerrail
      Contact( #BR12wAlm1.%X7 )
   END_RUNG wire#w1
   RUNG wire#powerrail
      Contact( #BR12wAlm1.%X8 )
   END_RUNG wire#w1
   RUNG wire#powerrail
      Contact( #BR12wAlm1.%X9 )
   END_RUNG wire#w1
   RUNG wire#powerrail
      Contact( #BR12wAlm1.%X10 )
   END_RUNG wire#w1
   RUNG wire#powerrail
      Contact( #BR12wAlm1.%X11 )
   END_RUNG wire#w1
   RUNG wire#powerrail
      Contact( #BR12wAlm1.%X12 )
   END_RUNG wire#w1
   RUNG wire#powerrail
      Contact( #BR12wAlm1.%X13 )
   END_RUNG wire#w1
   RUNG wire#powerrail
      Contact( #BR12wAlm3.%X0 )
   END_RUNG wire#w1
   RUNG wire#powerrail
      Contact( #BR12wAlm3.%X8 )
   END_RUNG wire#w1
   RUNG wire#powerrail
      Contact( #BR12wAlm3.%X9 )
   END_RUNG wire#w1
   // the same network as SCL:
   "BMS2".BR12xAlmSt := #BR12wAlm1.%X0 OR #BR12wAlm1.%X1 OR #BR12wAlm1.%X2 OR #BR12wAlm1.%X3 OR #BR12wAlm1.%X4 OR #BR12wAlm1.%X5 OR #BR12wAlm1.%X6 OR #BR12wAlm1.%X7 OR #BR12wAlm1.%X8 OR #BR12wAlm1.%X9 OR #BR12wAlm1.%X10 OR #BR12wAlm1.%X11 OR #BR12wAlm1.%X12 OR #BR12wAlm1.%X13 OR #BR12wAlm3.%X0 OR #BR12wAlm3.%X8 OR #BR12wAlm3.%X9;
END_REGION

REGION Network 124: BMS2 BR12 Warning
   RUNG wire#powerrail
      { S7_Templates := "SrcType := Word" } NE_Contact(in1 := #BR12wWarn1, in2 := 0)
      Coil( "BMS2".BR12xWarnSt )
   END_RUNG
   // the same network as SCL:
   "BMS2".BR12xWarnSt := #BR12wWarn1 <> 0;
END_REGION
END_FUNCTION

FUNCTION "Digital Output (comment out)" : Void   // FC5, LAD
{ S7_Optimized_Access := 'TRUE' }
VERSION : 0.1
// stored: AutoNumber false, IsIECCheckEnabled false, SetENOAutomatically false, UDAEnableTagReadback false
BEGIN

REGION Network 1: Digital Output 1
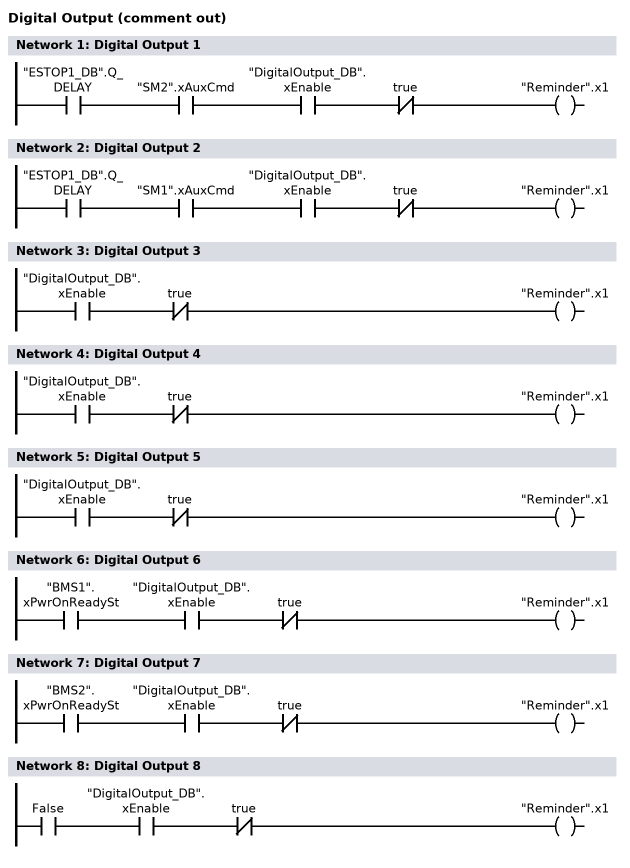
   RUNG wire#powerrail
      Contact( "ESTOP1_DB".Q_DELAY )
      Contact( "SM2".xAuxCmd )
      Contact( "DigitalOutput_DB".xEnable )
      I_Contact( true )
      Coil( "Reminder".x1 )
   END_RUNG
   // the same network as SCL:
   "Reminder".x1 := "ESTOP1_DB".Q_DELAY AND "SM2".xAuxCmd AND "DigitalOutput_DB".xEnable AND NOT true;
END_REGION

REGION Network 2: Digital Output 2
   RUNG wire#powerrail
      Contact( "ESTOP1_DB".Q_DELAY )
      Contact( "SM1".xAuxCmd )
      Contact( "DigitalOutput_DB".xEnable )
      I_Contact( true )
      Coil( "Reminder".x1 )
   END_RUNG
   // the same network as SCL:
   "Reminder".x1 := "ESTOP1_DB".Q_DELAY AND "SM1".xAuxCmd AND "DigitalOutput_DB".xEnable AND NOT true;
END_REGION

REGION Network 3: Digital Output 3
   RUNG wire#powerrail
      Contact( "DigitalOutput_DB".xEnable )
      I_Contact( true )
      Coil( "Reminder".x1 )
   END_RUNG
   // the same network as SCL:
   "Reminder".x1 := "DigitalOutput_DB".xEnable AND NOT true;
END_REGION

REGION Network 4: Digital Output 4
   RUNG wire#powerrail
      Contact( "DigitalOutput_DB".xEnable )
      I_Contact( true )
      Coil( "Reminder".x1 )
   END_RUNG
   // the same network as SCL:
   "Reminder".x1 := "DigitalOutput_DB".xEnable AND NOT true;
END_REGION

REGION Network 5: Digital Output 5
   RUNG wire#powerrail
      Contact( "DigitalOutput_DB".xEnable )
      I_Contact( true )
      Coil( "Reminder".x1 )
   END_RUNG
   // the same network as SCL:
   "Reminder".x1 := "DigitalOutput_DB".xEnable AND NOT true;
END_REGION

REGION Network 6: Digital Output 6
   RUNG wire#powerrail
      Contact( "BMS1".xPwrOnReadySt )
      Contact( "DigitalOutput_DB".xEnable )
      I_Contact( true )
      Coil( "Reminder".x1 )
   END_RUNG
   // the same network as SCL:
   "Reminder".x1 := "BMS1".xPwrOnReadySt AND "DigitalOutput_DB".xEnable AND NOT true;
END_REGION

REGION Network 7: Digital Output 7
   RUNG wire#powerrail
      Contact( "BMS2".xPwrOnReadySt )
      Contact( "DigitalOutput_DB".xEnable )
      I_Contact( true )
      Coil( "Reminder".x1 )
   END_RUNG
   // the same network as SCL:
   "Reminder".x1 := "BMS2".xPwrOnReadySt AND "DigitalOutput_DB".xEnable AND NOT true;
END_REGION

REGION Network 8: Digital Output 8
   RUNG wire#powerrail
      Contact( False )
      Contact( "DigitalOutput_DB".xEnable )
      I_Contact( true )
      Coil( "Reminder".x1 )
   END_RUNG
   // the same network as SCL:
   "Reminder".x1 := False AND "DigitalOutput_DB".xEnable AND NOT true;
END_REGION
END_FUNCTION

FUNCTION "AssetSt" : Void   // FC122, LAD
{ S7_Optimized_Access := 'TRUE' }
VERSION : 0.1
// stored: AutoNumber false, IsIECCheckEnabled false, SetENOAutomatically false, UDAEnableTagReadback false
BEGIN

REGION Network 1: Asset Status Battery Bank 1
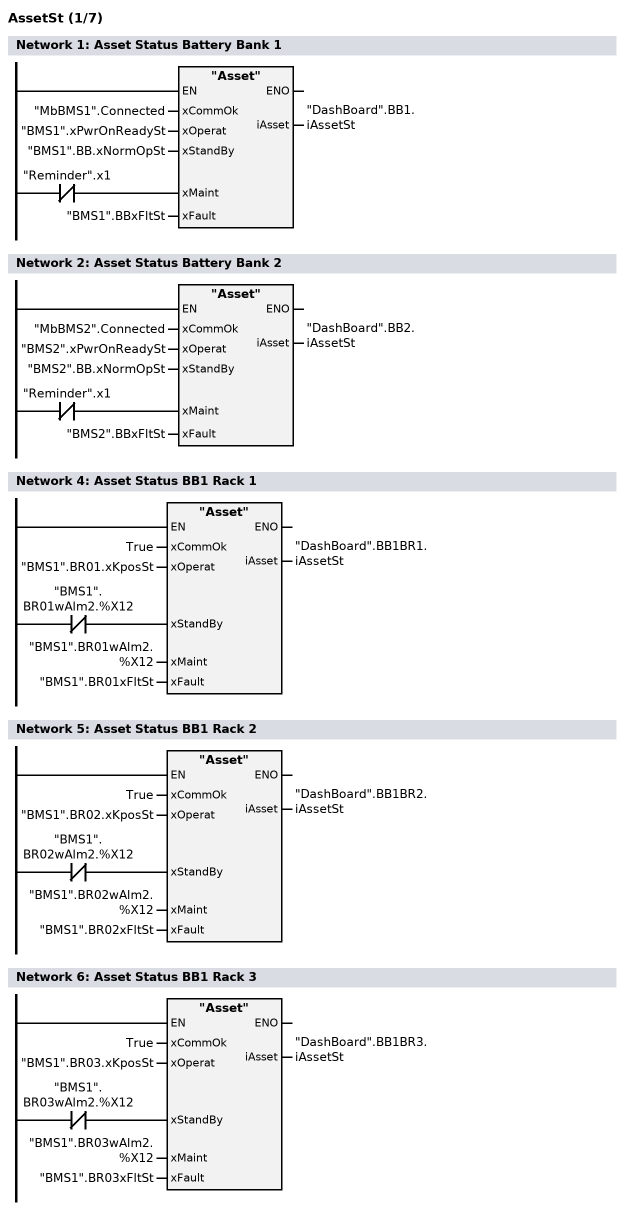
   RUNG wire#powerrail
      "Asset"(xMaint := wire#w1, xCommOk := "MbBMS1".Connected, xOperat := "BMS1".xPwrOnReadySt, xStandBy := "BMS1".BB.xNormOpSt, xFault := "BMS1".BBxFltSt, iAsset => "DashBoard".BB1.iAssetSt)
   END_RUNG
   RUNG wire#powerrail
      I_Contact( "Reminder".x1 )
   END_RUNG wire#w1
   // the same network as SCL:
   "Asset"(xCommOk := "MbBMS1".Connected,
           xOperat := "BMS1".xPwrOnReadySt,
           xStandBy := "BMS1".BB.xNormOpSt,
           xMaint := NOT "Reminder".x1,
           xFault := "BMS1".BBxFltSt,
           iAsset => "DashBoard".BB1.iAssetSt);
END_REGION

REGION Network 2: Asset Status Battery Bank 2
   RUNG wire#powerrail
      "Asset"(xMaint := wire#w1, xCommOk := "MbBMS2".Connected, xOperat := "BMS2".xPwrOnReadySt, xStandBy := "BMS2".BB.xNormOpSt, xFault := "BMS2".BBxFltSt, iAsset => "DashBoard".BB2.iAssetSt)
   END_RUNG
   RUNG wire#powerrail
      I_Contact( "Reminder".x1 )
   END_RUNG wire#w1
   // the same network as SCL:
   "Asset"(xCommOk := "MbBMS2".Connected,
           xOperat := "BMS2".xPwrOnReadySt,
           xStandBy := "BMS2".BB.xNormOpSt,
           xMaint := NOT "Reminder".x1,
           xFault := "BMS2".BBxFltSt,
           iAsset => "DashBoard".BB2.iAssetSt);
END_REGION

REGION Network 4: Asset Status BB1 Rack 1
   RUNG wire#powerrail
      "Asset"(xStandBy := wire#w1, xCommOk := True, xOperat := "BMS1".BR01.xKposSt, xMaint := "BMS1".BR01wAlm2.%X12, xFault := "BMS1".BR01xFltSt, iAsset => "DashBoard".BB1BR1.iAssetSt)
   END_RUNG
   RUNG wire#powerrail
      I_Contact( "BMS1".BR01wAlm2.%X12 )
   END_RUNG wire#w1
   // the same network as SCL:
   "Asset"(xCommOk := True,
           xOperat := "BMS1".BR01.xKposSt,
           xStandBy := NOT "BMS1".BR01wAlm2.%X12,
           xMaint := "BMS1".BR01wAlm2.%X12,
           xFault := "BMS1".BR01xFltSt,
           iAsset => "DashBoard".BB1BR1.iAssetSt);
END_REGION

REGION Network 5: Asset Status BB1 Rack 2
   RUNG wire#powerrail
      "Asset"(xStandBy := wire#w1, xCommOk := True, xOperat := "BMS1".BR02.xKposSt, xMaint := "BMS1".BR02wAlm2.%X12, xFault := "BMS1".BR02xFltSt, iAsset => "DashBoard".BB1BR2.iAssetSt)
   END_RUNG
   RUNG wire#powerrail
      I_Contact( "BMS1".BR02wAlm2.%X12 )
   END_RUNG wire#w1
   // the same network as SCL:
   "Asset"(xCommOk := True,
           xOperat := "BMS1".BR02.xKposSt,
           xStandBy := NOT "BMS1".BR02wAlm2.%X12,
           xMaint := "BMS1".BR02wAlm2.%X12,
           xFault := "BMS1".BR02xFltSt,
           iAsset => "DashBoard".BB1BR2.iAssetSt);
END_REGION

REGION Network 6: Asset Status BB1 Rack 3
   RUNG wire#powerrail
      "Asset"(xStandBy := wire#w1, xCommOk := True, xOperat := "BMS1".BR03.xKposSt, xMaint := "BMS1".BR03wAlm2.%X12, xFault := "BMS1".BR03xFltSt, iAsset => "DashBoard".BB1BR3.iAssetSt)
   END_RUNG
   RUNG wire#powerrail
      I_Contact( "BMS1".BR03wAlm2.%X12 )
   END_RUNG wire#w1
   // the same network as SCL:
   "Asset"(xCommOk := True,
           xOperat := "BMS1".BR03.xKposSt,
           xStandBy := NOT "BMS1".BR03wAlm2.%X12,
           xMaint := "BMS1".BR03wAlm2.%X12,
           xFault := "BMS1".BR03xFltSt,
           iAsset => "DashBoard".BB1BR3.iAssetSt);
END_REGION

REGION Network 7: Asset Status BB1 Rack 4
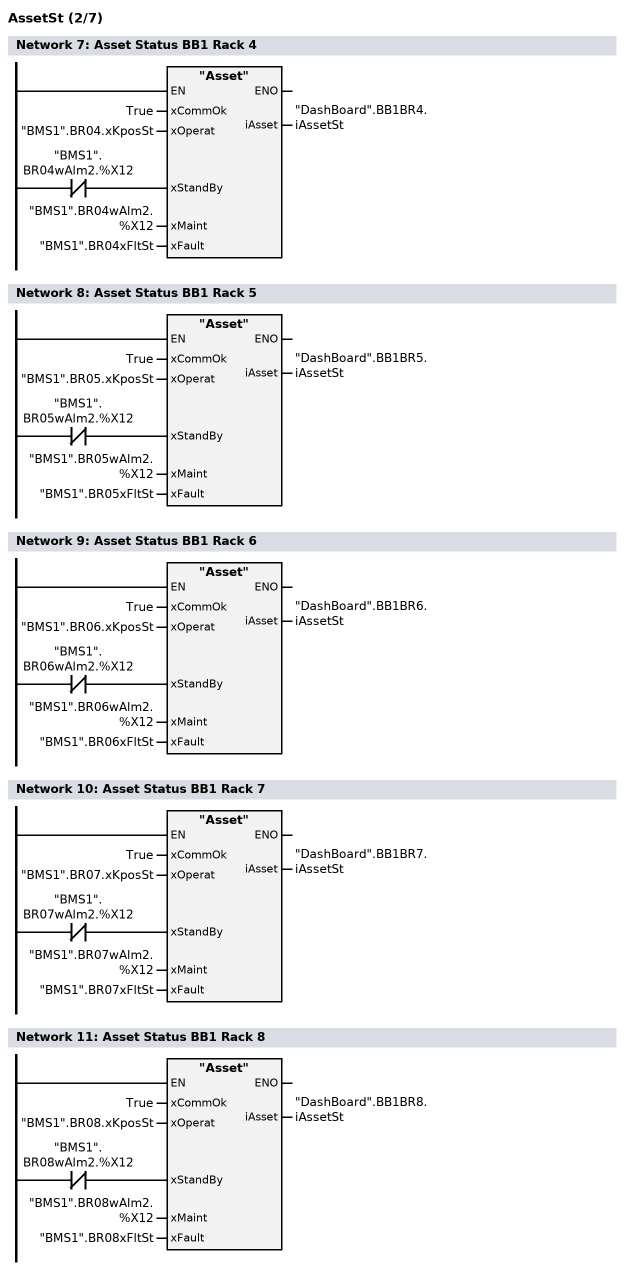
   RUNG wire#powerrail
      "Asset"(xStandBy := wire#w1, xCommOk := True, xOperat := "BMS1".BR04.xKposSt, xMaint := "BMS1".BR04wAlm2.%X12, xFault := "BMS1".BR04xFltSt, iAsset => "DashBoard".BB1BR4.iAssetSt)
   END_RUNG
   RUNG wire#powerrail
      I_Contact( "BMS1".BR04wAlm2.%X12 )
   END_RUNG wire#w1
   // the same network as SCL:
   "Asset"(xCommOk := True,
           xOperat := "BMS1".BR04.xKposSt,
           xStandBy := NOT "BMS1".BR04wAlm2.%X12,
           xMaint := "BMS1".BR04wAlm2.%X12,
           xFault := "BMS1".BR04xFltSt,
           iAsset => "DashBoard".BB1BR4.iAssetSt);
END_REGION

REGION Network 8: Asset Status BB1 Rack 5
   RUNG wire#powerrail
      "Asset"(xStandBy := wire#w1, xCommOk := True, xOperat := "BMS1".BR05.xKposSt, xMaint := "BMS1".BR05wAlm2.%X12, xFault := "BMS1".BR05xFltSt, iAsset => "DashBoard".BB1BR5.iAssetSt)
   END_RUNG
   RUNG wire#powerrail
      I_Contact( "BMS1".BR05wAlm2.%X12 )
   END_RUNG wire#w1
   // the same network as SCL:
   "Asset"(xCommOk := True,
           xOperat := "BMS1".BR05.xKposSt,
           xStandBy := NOT "BMS1".BR05wAlm2.%X12,
           xMaint := "BMS1".BR05wAlm2.%X12,
           xFault := "BMS1".BR05xFltSt,
           iAsset => "DashBoard".BB1BR5.iAssetSt);
END_REGION

REGION Network 9: Asset Status BB1 Rack 6
   RUNG wire#powerrail
      "Asset"(xStandBy := wire#w1, xCommOk := True, xOperat := "BMS1".BR06.xKposSt, xMaint := "BMS1".BR06wAlm2.%X12, xFault := "BMS1".BR06xFltSt, iAsset => "DashBoard".BB1BR6.iAssetSt)
   END_RUNG
   RUNG wire#powerrail
      I_Contact( "BMS1".BR06wAlm2.%X12 )
   END_RUNG wire#w1
   // the same network as SCL:
   "Asset"(xCommOk := True,
           xOperat := "BMS1".BR06.xKposSt,
           xStandBy := NOT "BMS1".BR06wAlm2.%X12,
           xMaint := "BMS1".BR06wAlm2.%X12,
           xFault := "BMS1".BR06xFltSt,
           iAsset => "DashBoard".BB1BR6.iAssetSt);
END_REGION

REGION Network 10: Asset Status BB1 Rack 7
   RUNG wire#powerrail
      "Asset"(xStandBy := wire#w1, xCommOk := True, xOperat := "BMS1".BR07.xKposSt, xMaint := "BMS1".BR07wAlm2.%X12, xFault := "BMS1".BR07xFltSt, iAsset => "DashBoard".BB1BR7.iAssetSt)
   END_RUNG
   RUNG wire#powerrail
      I_Contact( "BMS1".BR07wAlm2.%X12 )
   END_RUNG wire#w1
   // the same network as SCL:
   "Asset"(xCommOk := True,
           xOperat := "BMS1".BR07.xKposSt,
           xStandBy := NOT "BMS1".BR07wAlm2.%X12,
           xMaint := "BMS1".BR07wAlm2.%X12,
           xFault := "BMS1".BR07xFltSt,
           iAsset => "DashBoard".BB1BR7.iAssetSt);
END_REGION

REGION Network 11: Asset Status BB1 Rack 8
   RUNG wire#powerrail
      "Asset"(xStandBy := wire#w1, xCommOk := True, xOperat := "BMS1".BR08.xKposSt, xMaint := "BMS1".BR08wAlm2.%X12, xFault := "BMS1".BR08xFltSt, iAsset => "DashBoard".BB1BR8.iAssetSt)
   END_RUNG
   RUNG wire#powerrail
      I_Contact( "BMS1".BR08wAlm2.%X12 )
   END_RUNG wire#w1
   // the same network as SCL:
   "Asset"(xCommOk := True,
           xOperat := "BMS1".BR08.xKposSt,
           xStandBy := NOT "BMS1".BR08wAlm2.%X12,
           xMaint := "BMS1".BR08wAlm2.%X12,
           xFault := "BMS1".BR08xFltSt,
           iAsset => "DashBoard".BB1BR8.iAssetSt);
END_REGION

REGION Network 12: Asset Status BB1 Rack 9
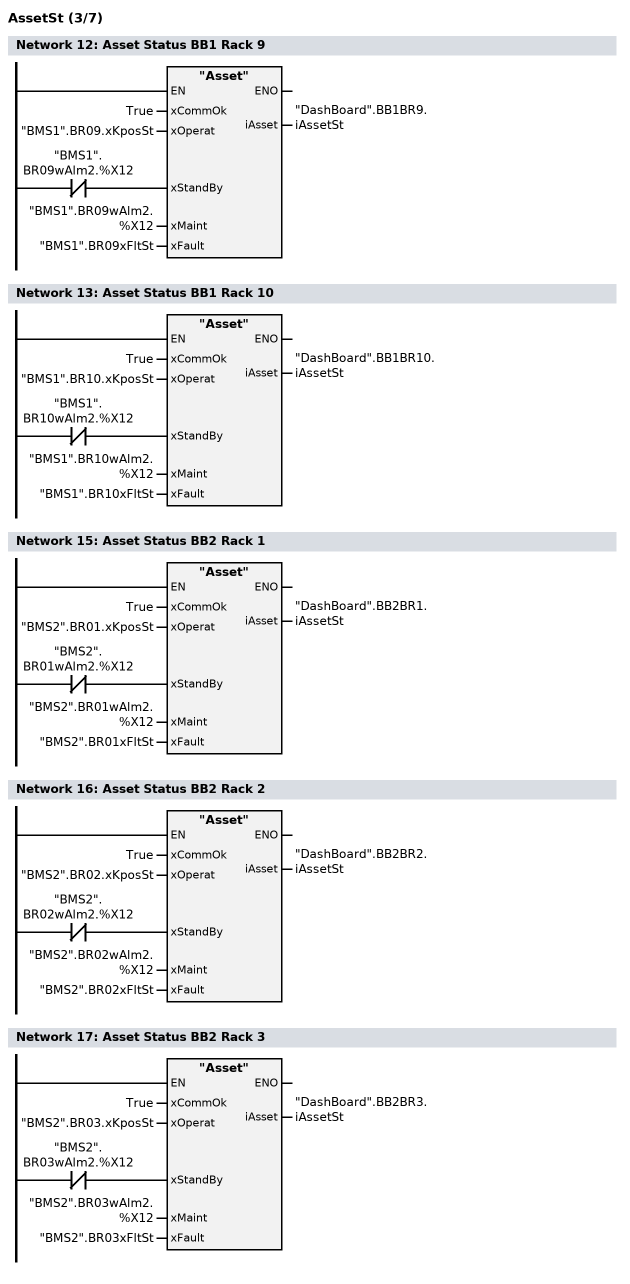
   RUNG wire#powerrail
      "Asset"(xStandBy := wire#w1, xCommOk := True, xOperat := "BMS1".BR09.xKposSt, xMaint := "BMS1".BR09wAlm2.%X12, xFault := "BMS1".BR09xFltSt, iAsset => "DashBoard".BB1BR9.iAssetSt)
   END_RUNG
   RUNG wire#powerrail
      I_Contact( "BMS1".BR09wAlm2.%X12 )
   END_RUNG wire#w1
   // the same network as SCL:
   "Asset"(xCommOk := True,
           xOperat := "BMS1".BR09.xKposSt,
           xStandBy := NOT "BMS1".BR09wAlm2.%X12,
           xMaint := "BMS1".BR09wAlm2.%X12,
           xFault := "BMS1".BR09xFltSt,
           iAsset => "DashBoard".BB1BR9.iAssetSt);
END_REGION

REGION Network 13: Asset Status BB1 Rack 10
   RUNG wire#powerrail
      "Asset"(xStandBy := wire#w1, xCommOk := True, xOperat := "BMS1".BR10.xKposSt, xMaint := "BMS1".BR10wAlm2.%X12, xFault := "BMS1".BR10xFltSt, iAsset => "DashBoard".BB1BR10.iAssetSt)
   END_RUNG
   RUNG wire#powerrail
      I_Contact( "BMS1".BR10wAlm2.%X12 )
   END_RUNG wire#w1
   // the same network as SCL:
   "Asset"(xCommOk := True,
           xOperat := "BMS1".BR10.xKposSt,
           xStandBy := NOT "BMS1".BR10wAlm2.%X12,
           xMaint := "BMS1".BR10wAlm2.%X12,
           xFault := "BMS1".BR10xFltSt,
           iAsset => "DashBoard".BB1BR10.iAssetSt);
END_REGION

REGION Network 15: Asset Status BB2 Rack 1
   RUNG wire#powerrail
      "Asset"(xStandBy := wire#w1, xCommOk := True, xOperat := "BMS2".BR01.xKposSt, xMaint := "BMS2".BR01wAlm2.%X12, xFault := "BMS2".BR01xFltSt, iAsset => "DashBoard".BB2BR1.iAssetSt)
   END_RUNG
   RUNG wire#powerrail
      I_Contact( "BMS2".BR01wAlm2.%X12 )
   END_RUNG wire#w1
   // the same network as SCL:
   "Asset"(xCommOk := True,
           xOperat := "BMS2".BR01.xKposSt,
           xStandBy := NOT "BMS2".BR01wAlm2.%X12,
           xMaint := "BMS2".BR01wAlm2.%X12,
           xFault := "BMS2".BR01xFltSt,
           iAsset => "DashBoard".BB2BR1.iAssetSt);
END_REGION

REGION Network 16: Asset Status BB2 Rack 2
   RUNG wire#powerrail
      "Asset"(xStandBy := wire#w1, xCommOk := True, xOperat := "BMS2".BR02.xKposSt, xMaint := "BMS2".BR02wAlm2.%X12, xFault := "BMS2".BR02xFltSt, iAsset => "DashBoard".BB2BR2.iAssetSt)
   END_RUNG
   RUNG wire#powerrail
      I_Contact( "BMS2".BR02wAlm2.%X12 )
   END_RUNG wire#w1
   // the same network as SCL:
   "Asset"(xCommOk := True,
           xOperat := "BMS2".BR02.xKposSt,
           xStandBy := NOT "BMS2".BR02wAlm2.%X12,
           xMaint := "BMS2".BR02wAlm2.%X12,
           xFault := "BMS2".BR02xFltSt,
           iAsset => "DashBoard".BB2BR2.iAssetSt);
END_REGION

REGION Network 17: Asset Status BB2 Rack 3
   RUNG wire#powerrail
      "Asset"(xStandBy := wire#w1, xCommOk := True, xOperat := "BMS2".BR03.xKposSt, xMaint := "BMS2".BR03wAlm2.%X12, xFault := "BMS2".BR03xFltSt, iAsset => "DashBoard".BB2BR3.iAssetSt)
   END_RUNG
   RUNG wire#powerrail
      I_Contact( "BMS2".BR03wAlm2.%X12 )
   END_RUNG wire#w1
   // the same network as SCL:
   "Asset"(xCommOk := True,
           xOperat := "BMS2".BR03.xKposSt,
           xStandBy := NOT "BMS2".BR03wAlm2.%X12,
           xMaint := "BMS2".BR03wAlm2.%X12,
           xFault := "BMS2".BR03xFltSt,
           iAsset => "DashBoard".BB2BR3.iAssetSt);
END_REGION

REGION Network 18: Asset Status BB2 Rack 4
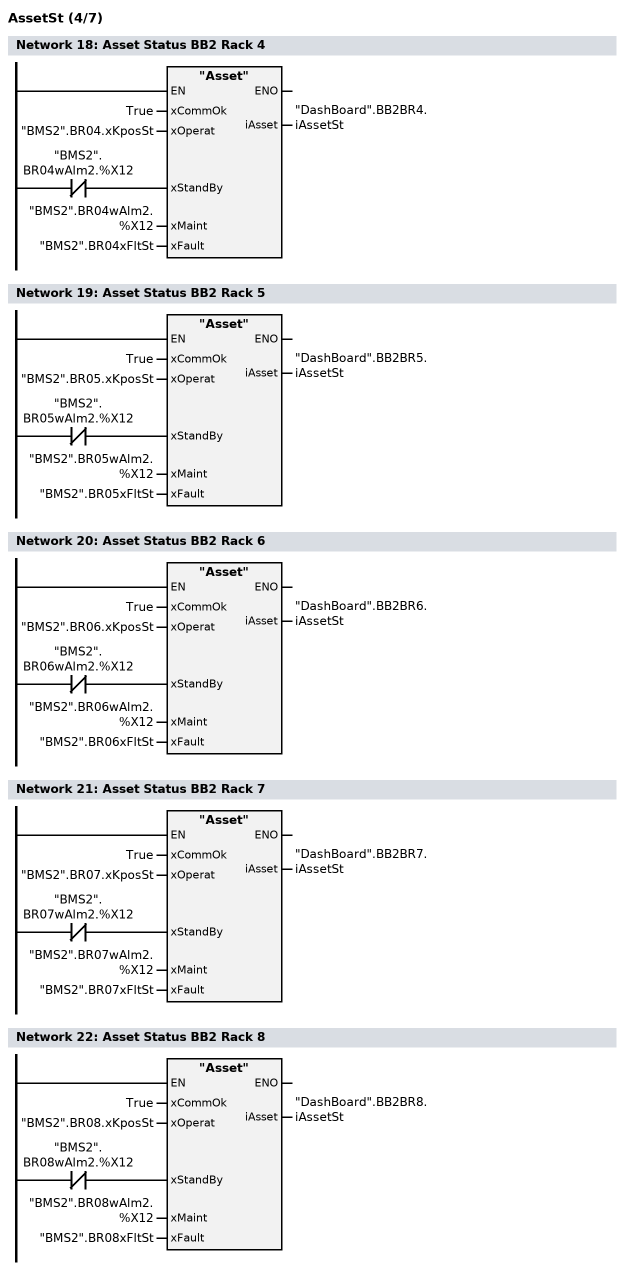
   RUNG wire#powerrail
      "Asset"(xStandBy := wire#w1, xCommOk := True, xOperat := "BMS2".BR04.xKposSt, xMaint := "BMS2".BR04wAlm2.%X12, xFault := "BMS2".BR04xFltSt, iAsset => "DashBoard".BB2BR4.iAssetSt)
   END_RUNG
   RUNG wire#powerrail
      I_Contact( "BMS2".BR04wAlm2.%X12 )
   END_RUNG wire#w1
   // the same network as SCL:
   "Asset"(xCommOk := True,
           xOperat := "BMS2".BR04.xKposSt,
           xStandBy := NOT "BMS2".BR04wAlm2.%X12,
           xMaint := "BMS2".BR04wAlm2.%X12,
           xFault := "BMS2".BR04xFltSt,
           iAsset => "DashBoard".BB2BR4.iAssetSt);
END_REGION

REGION Network 19: Asset Status BB2 Rack 5
   RUNG wire#powerrail
      "Asset"(xStandBy := wire#w1, xCommOk := True, xOperat := "BMS2".BR05.xKposSt, xMaint := "BMS2".BR05wAlm2.%X12, xFault := "BMS2".BR05xFltSt, iAsset => "DashBoard".BB2BR5.iAssetSt)
   END_RUNG
   RUNG wire#powerrail
      I_Contact( "BMS2".BR05wAlm2.%X12 )
   END_RUNG wire#w1
   // the same network as SCL:
   "Asset"(xCommOk := True,
           xOperat := "BMS2".BR05.xKposSt,
           xStandBy := NOT "BMS2".BR05wAlm2.%X12,
           xMaint := "BMS2".BR05wAlm2.%X12,
           xFault := "BMS2".BR05xFltSt,
           iAsset => "DashBoard".BB2BR5.iAssetSt);
END_REGION

REGION Network 20: Asset Status BB2 Rack 6
   RUNG wire#powerrail
      "Asset"(xStandBy := wire#w1, xCommOk := True, xOperat := "BMS2".BR06.xKposSt, xMaint := "BMS2".BR06wAlm2.%X12, xFault := "BMS2".BR06xFltSt, iAsset => "DashBoard".BB2BR6.iAssetSt)
   END_RUNG
   RUNG wire#powerrail
      I_Contact( "BMS2".BR06wAlm2.%X12 )
   END_RUNG wire#w1
   // the same network as SCL:
   "Asset"(xCommOk := True,
           xOperat := "BMS2".BR06.xKposSt,
           xStandBy := NOT "BMS2".BR06wAlm2.%X12,
           xMaint := "BMS2".BR06wAlm2.%X12,
           xFault := "BMS2".BR06xFltSt,
           iAsset => "DashBoard".BB2BR6.iAssetSt);
END_REGION

REGION Network 21: Asset Status BB2 Rack 7
   RUNG wire#powerrail
      "Asset"(xStandBy := wire#w1, xCommOk := True, xOperat := "BMS2".BR07.xKposSt, xMaint := "BMS2".BR07wAlm2.%X12, xFault := "BMS2".BR07xFltSt, iAsset => "DashBoard".BB2BR7.iAssetSt)
   END_RUNG
   RUNG wire#powerrail
      I_Contact( "BMS2".BR07wAlm2.%X12 )
   END_RUNG wire#w1
   // the same network as SCL:
   "Asset"(xCommOk := True,
           xOperat := "BMS2".BR07.xKposSt,
           xStandBy := NOT "BMS2".BR07wAlm2.%X12,
           xMaint := "BMS2".BR07wAlm2.%X12,
           xFault := "BMS2".BR07xFltSt,
           iAsset => "DashBoard".BB2BR7.iAssetSt);
END_REGION

REGION Network 22: Asset Status BB2 Rack 8
   RUNG wire#powerrail
      "Asset"(xStandBy := wire#w1, xCommOk := True, xOperat := "BMS2".BR08.xKposSt, xMaint := "BMS2".BR08wAlm2.%X12, xFault := "BMS2".BR08xFltSt, iAsset => "DashBoard".BB2BR8.iAssetSt)
   END_RUNG
   RUNG wire#powerrail
      I_Contact( "BMS2".BR08wAlm2.%X12 )
   END_RUNG wire#w1
   // the same network as SCL:
   "Asset"(xCommOk := True,
           xOperat := "BMS2".BR08.xKposSt,
           xStandBy := NOT "BMS2".BR08wAlm2.%X12,
           xMaint := "BMS2".BR08wAlm2.%X12,
           xFault := "BMS2".BR08xFltSt,
           iAsset => "DashBoard".BB2BR8.iAssetSt);
END_REGION

REGION Network 23: Asset Status BB2 Rack 9
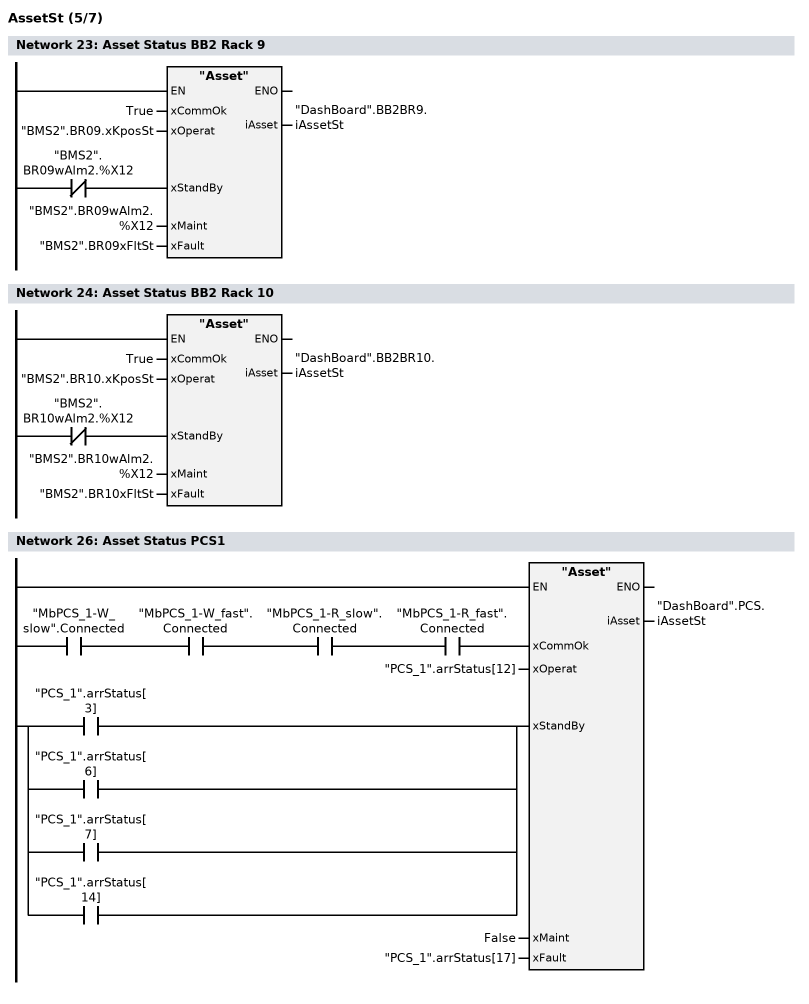
   RUNG wire#powerrail
      "Asset"(xStandBy := wire#w1, xCommOk := True, xOperat := "BMS2".BR09.xKposSt, xMaint := "BMS2".BR09wAlm2.%X12, xFault := "BMS2".BR09xFltSt, iAsset => "DashBoard".BB2BR9.iAssetSt)
   END_RUNG
   RUNG wire#powerrail
      I_Contact( "BMS2".BR09wAlm2.%X12 )
   END_RUNG wire#w1
   // the same network as SCL:
   "Asset"(xCommOk := True,
           xOperat := "BMS2".BR09.xKposSt,
           xStandBy := NOT "BMS2".BR09wAlm2.%X12,
           xMaint := "BMS2".BR09wAlm2.%X12,
           xFault := "BMS2".BR09xFltSt,
           iAsset => "DashBoard".BB2BR9.iAssetSt);
END_REGION

REGION Network 24: Asset Status BB2 Rack 10
   RUNG wire#powerrail
      "Asset"(xStandBy := wire#w1, xCommOk := True, xOperat := "BMS2".BR10.xKposSt, xMaint := "BMS2".BR10wAlm2.%X12, xFault := "BMS2".BR10xFltSt, iAsset => "DashBoard".BB2BR10.iAssetSt)
   END_RUNG
   RUNG wire#powerrail
      I_Contact( "BMS2".BR10wAlm2.%X12 )
   END_RUNG wire#w1
   // the same network as SCL:
   "Asset"(xCommOk := True,
           xOperat := "BMS2".BR10.xKposSt,
           xStandBy := NOT "BMS2".BR10wAlm2.%X12,
           xMaint := "BMS2".BR10wAlm2.%X12,
           xFault := "BMS2".BR10xFltSt,
           iAsset => "DashBoard".BB2BR10.iAssetSt);
END_REGION

REGION Network 26: Asset Status PCS1
   RUNG wire#powerrail
      "Asset"(xCommOk := wire#w1, xStandBy := wire#w2, xOperat := "PCS_1".arrStatus[12], xMaint := False, xFault := "PCS_1".arrStatus[17], iAsset => "DashBoard".PCS.iAssetSt)
   END_RUNG
   RUNG wire#powerrail
      Contact( "MbPCS_1-W_slow".Connected )
      Contact( "MbPCS_1-W_fast".Connected )
      Contact( "MbPCS_1-R_slow".Connected )
      Contact( "MbPCS_1-R_fast".Connected )
   END_RUNG wire#w1
   RUNG wire#powerrail
      Contact( "PCS_1".arrStatus[3] )
   END_RUNG wire#w2
   RUNG wire#powerrail
      Contact( "PCS_1".arrStatus[6] )
   END_RUNG wire#w2
   RUNG wire#powerrail
      Contact( "PCS_1".arrStatus[7] )
   END_RUNG wire#w2
   RUNG wire#powerrail
      Contact( "PCS_1".arrStatus[14] )
   END_RUNG wire#w2
   // the same network as SCL:
   "Asset"(xCommOk := "MbPCS_1-W_slow".Connected AND "MbPCS_1-W_fast".Connected AND "MbPCS_1-R_slow".Connected AND "MbPCS_1-R_fast".Connected,
           xOperat := "PCS_1".arrStatus[12],
           xStandBy := "PCS_1".arrStatus[3] OR "PCS_1".arrStatus[6] OR "PCS_1".arrStatus[7] OR "PCS_1".arrStatus[14],
           xMaint := False,
           xFault := "PCS_1".arrStatus[17],
           iAsset => "DashBoard".PCS.iAssetSt);
END_REGION

REGION Network 27: Asset Status PCS1
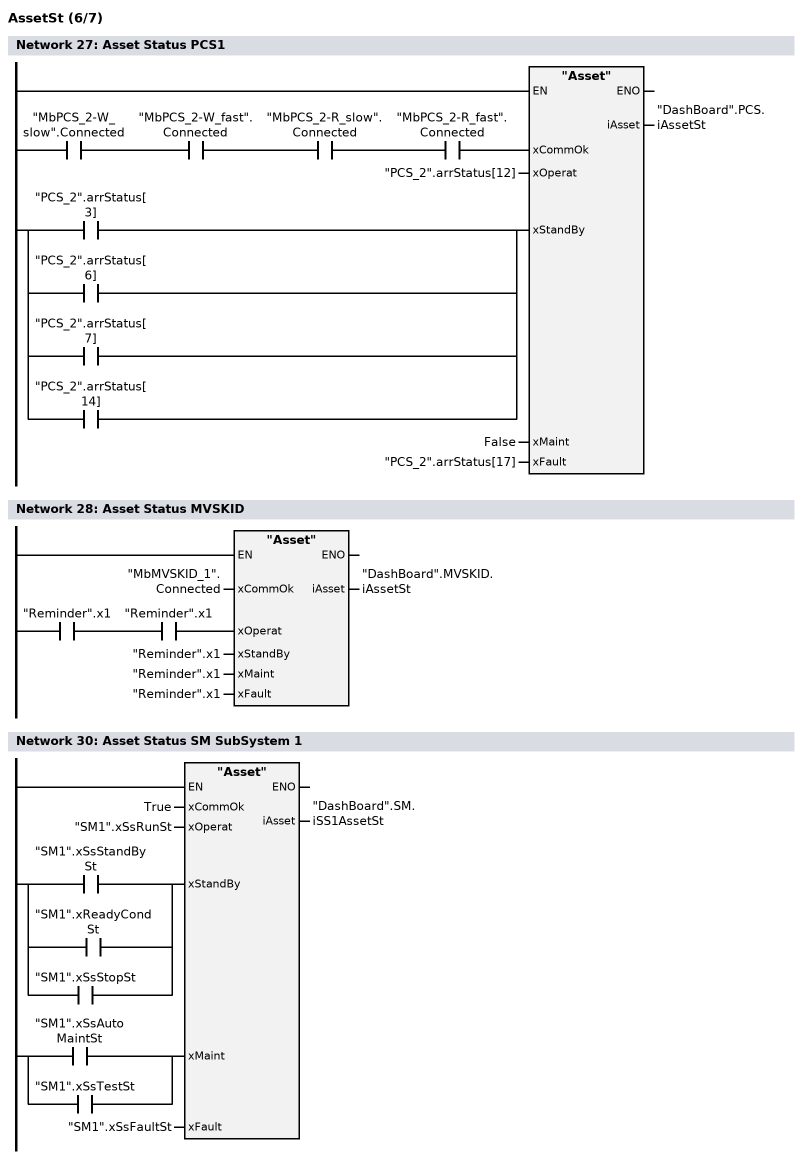
   RUNG wire#powerrail
      "Asset"(xCommOk := wire#w1, xStandBy := wire#w2, xOperat := "PCS_2".arrStatus[12], xMaint := False, xFault := "PCS_2".arrStatus[17], iAsset => "DashBoard".PCS.iAssetSt)
   END_RUNG
   RUNG wire#powerrail
      Contact( "MbPCS_2-W_slow".Connected )
      Contact( "MbPCS_2-W_fast".Connected )
      Contact( "MbPCS_2-R_slow".Connected )
      Contact( "MbPCS_2-R_fast".Connected )
   END_RUNG wire#w1
   RUNG wire#powerrail
      Contact( "PCS_2".arrStatus[3] )
   END_RUNG wire#w2
   RUNG wire#powerrail
      Contact( "PCS_2".arrStatus[6] )
   END_RUNG wire#w2
   RUNG wire#powerrail
      Contact( "PCS_2".arrStatus[7] )
   END_RUNG wire#w2
   RUNG wire#powerrail
      Contact( "PCS_2".arrStatus[14] )
   END_RUNG wire#w2
   // the same network as SCL:
   "Asset"(xCommOk := "MbPCS_2-W_slow".Connected AND "MbPCS_2-W_fast".Connected AND "MbPCS_2-R_slow".Connected AND "MbPCS_2-R_fast".Connected,
           xOperat := "PCS_2".arrStatus[12],
           xStandBy := "PCS_2".arrStatus[3] OR "PCS_2".arrStatus[6] OR "PCS_2".arrStatus[7] OR "PCS_2".arrStatus[14],
           xMaint := False,
           xFault := "PCS_2".arrStatus[17],
           iAsset => "DashBoard".PCS.iAssetSt);
END_REGION

REGION Network 28: Asset Status MVSKID
   RUNG wire#powerrail
      "Asset"(xOperat := wire#w1, xCommOk := "MbMVSKID_1".Connected, xStandBy := "Reminder".x1, xMaint := "Reminder".x1, xFault := "Reminder".x1, iAsset => "DashBoard".MVSKID.iAssetSt)
   END_RUNG
   RUNG wire#powerrail
      Contact( "Reminder".x1 )
      Contact( "Reminder".x1 )
   END_RUNG wire#w1
   // the same network as SCL:
   "Asset"(xCommOk := "MbMVSKID_1".Connected,
           xOperat := "Reminder".x1 AND "Reminder".x1,
           xStandBy := "Reminder".x1,
           xMaint := "Reminder".x1,
           xFault := "Reminder".x1,
           iAsset => "DashBoard".MVSKID.iAssetSt);
END_REGION

REGION Network 30: Asset Status SM SubSystem 1
   RUNG wire#powerrail
      "Asset"(xStandBy := wire#w1, xMaint := wire#w2, xCommOk := True, xOperat := "SM1".xSsRunSt, xFault := "SM1".xSsFaultSt, iAsset => "DashBoard".SM.iSS1AssetSt)
   END_RUNG
   RUNG wire#powerrail
      Contact( "SM1".xSsStandBySt )
   END_RUNG wire#w1
   RUNG wire#powerrail
      Contact( "SM1".xReadyCondSt )
   END_RUNG wire#w1
   RUNG wire#powerrail
      Contact( "SM1".xSsStopSt )
   END_RUNG wire#w1
   RUNG wire#powerrail
      Contact( "SM1".xSsAutoMaintSt )
   END_RUNG wire#w2
   RUNG wire#powerrail
      Contact( "SM1".xSsTestSt )
   END_RUNG wire#w2
   // the same network as SCL:
   "Asset"(xCommOk := True,
           xOperat := "SM1".xSsRunSt,
           xStandBy := "SM1".xSsStandBySt OR "SM1".xReadyCondSt OR "SM1".xSsStopSt,
           xMaint := "SM1".xSsAutoMaintSt OR "SM1".xSsTestSt,
           xFault := "SM1".xSsFaultSt,
           iAsset => "DashBoard".SM.iSS1AssetSt);
END_REGION

REGION Network 31: Asset Status SM SubSystem 2
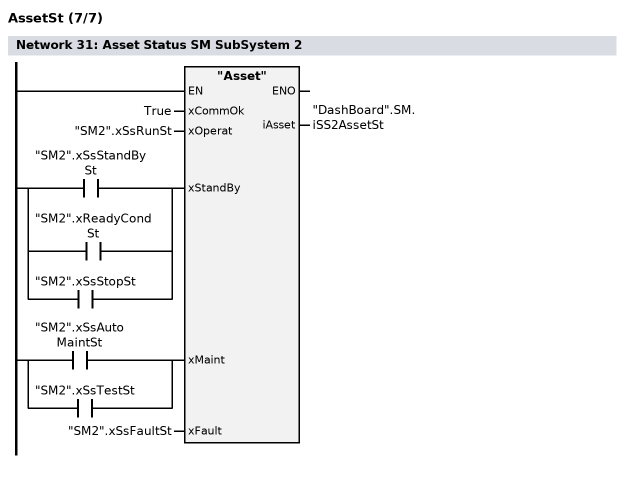
   RUNG wire#powerrail
      "Asset"(xStandBy := wire#w1, xMaint := wire#w2, xCommOk := True, xOperat := "SM2".xSsRunSt, xFault := "SM2".xSsFaultSt, iAsset => "DashBoard".SM.iSS2AssetSt)
   END_RUNG
   RUNG wire#powerrail
      Contact( "SM2".xSsStandBySt )
   END_RUNG wire#w1
   RUNG wire#powerrail
      Contact( "SM2".xReadyCondSt )
   END_RUNG wire#w1
   RUNG wire#powerrail
      Contact( "SM2".xSsStopSt )
   END_RUNG wire#w1
   RUNG wire#powerrail
      Contact( "SM2".xSsAutoMaintSt )
   END_RUNG wire#w2
   RUNG wire#powerrail
      Contact( "SM2".xSsTestSt )
   END_RUNG wire#w2
   // the same network as SCL:
   "Asset"(xCommOk := True,
           xOperat := "SM2".xSsRunSt,
           xStandBy := "SM2".xSsStandBySt OR "SM2".xReadyCondSt OR "SM2".xSsStopSt,
           xMaint := "SM2".xSsAutoMaintSt OR "SM2".xSsTestSt,
           xFault := "SM2".xSsFaultSt,
           iAsset => "DashBoard".SM.iSS2AssetSt);
END_REGION
END_FUNCTION

FUNCTION "Asset" : Void
{ S7_Optimized_Access := 'TRUE' }
VERSION : 0.1
   VAR_INPUT 
      xCommOk : Bool;
      xOperat : Bool;
      xStandBy : Bool;
      xMaint : Bool;
      xFault : Bool;
   END_VAR

   VAR_OUTPUT 
      iAsset : Int;
   END_VAR


BEGIN
	
	IF #xCommOk
	THEN
	    
	    IF #xOperat
	    THEN
	        #iAsset := 1;
	    ELSIF #xStandBy
	    THEN
	        #iAsset := 2;
	    ELSIF #xMaint
	    THEN
	        #iAsset := 3;
	    ELSIF #xFault
	    THEN
	        #iAsset := 4;
	    ELSE
	        #iAsset := 0;
	    END_IF;
	    
	ELSE
	    #iAsset := 0;
	END_IF;
	
END_FUNCTION

FUNCTION "EthernetDiag" : Void   // FC401, LAD
TITLE = Ethernet Diagnostic
{ S7_Optimized_Access := 'TRUE' }
VERSION : 0.1
// stored: AutoNumber false, IsIECCheckEnabled false, SetENOAutomatically false, UDAEnableTagReadback false
BEGIN

REGION Network 1: Ethernet Diagnostic PLC PEMS
   // Block to check ethernet connection to PEMS (used in HMI)
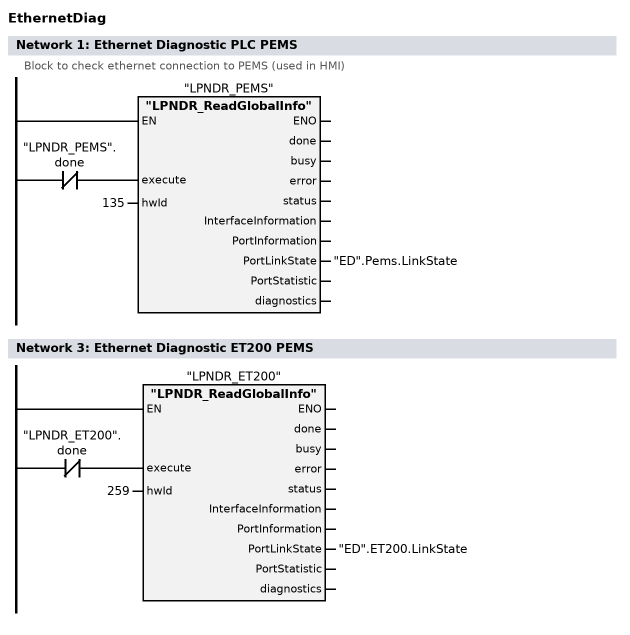
   RUNG wire#powerrail
      "LPNDR_PEMS"(execute := wire#w1, hwId := 135, done =>, busy =>, error =>, status =>, InterfaceInformation =>, PortInformation =>, PortLinkState => "ED".Pems.LinkState, PortStatistic =>, diagnostics =>)
   END_RUNG
   RUNG wire#powerrail
      I_Contact( "LPNDR_PEMS".done )
   END_RUNG wire#w1
   // the same network as SCL:
   "LPNDR_PEMS"(execute := NOT "LPNDR_PEMS".done, hwId := 135, PortLinkState => "ED".Pems.LinkState);   // "LPNDR_ReadGlobalInfo"
END_REGION

REGION Network 2 (SCL): Ethernet Diagnostic PLC PEMS
   "ED".Pems.X1 := "ED".Pems.LinkState[1].portLinkState = 1;
   "ED".Pems.X2 := "ED".Pems.LinkState[2].portLinkState = 1;
   "ED".Pems.X3 := "ED".Pems.LinkState[3].portLinkState = 1;
END_REGION

REGION Network 3: Ethernet Diagnostic ET200 PEMS
   RUNG wire#powerrail
      "LPNDR_ET200"(execute := wire#w1, hwId := 259, done =>, busy =>, error =>, status =>, InterfaceInformation =>, PortInformation =>, PortLinkState => "ED".ET200.LinkState, PortStatistic =>, diagnostics =>)
   END_RUNG
   RUNG wire#powerrail
      I_Contact( "LPNDR_ET200".done )
   END_RUNG wire#w1
   // the same network as SCL:
   "LPNDR_ET200"(execute := NOT "LPNDR_ET200".done, hwId := 259, PortLinkState => "ED".ET200.LinkState);   // "LPNDR_ReadGlobalInfo"
END_REGION

REGION Network 4 (SCL): Ethernet Diagnostic ET200 PEMS
   "ED".ET200.X1 := "ED".ET200.LinkState[1].portLinkState = 1;
   "ED".ET200.X2 := "ED".ET200.LinkState[2].portLinkState = 1;
END_REGION
END_FUNCTION

FUNCTION "NTP" : Void   // FC124, LAD
{ S7_Optimized_Access := 'TRUE' }
VERSION : 0.1
// stored: AutoNumber false, IsIECCheckEnabled false, SetENOAutomatically false, UDAEnableTagReadback false
   VAR_TEMP   // added for the SCL form of the ladder/FBD networks
      _w1 : Bool;
   END_VAR
BEGIN

REGION Network 1: Server NTP
   // To run also in a task 1s, it's used by the MINI_PC to retrieve the correct date and time
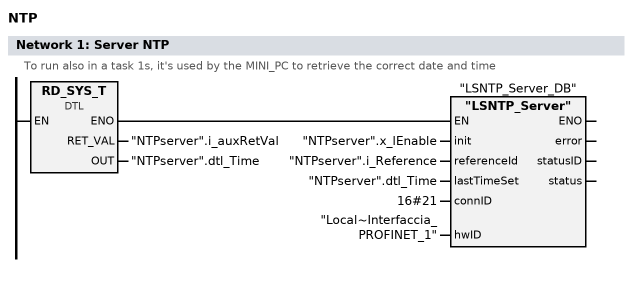
   RUNG wire#powerrail
      { S7_Templates := "date_type := DTL" } RD_SYS_T(RET_VAL => "NTPserver".i_auxRetVal, OUT => "NTPserver".dtl_Time)
      "LSNTP_Server_DB"(init := "NTPserver".x_lEnable, referenceId := "NTPserver".i_Reference, lastTimeSet := "NTPserver".dtl_Time, connID := 16#21, hwID := "Local~Interfaccia_PROFINET_1", error =>, statusID =>, status =>)
   END_RUNG
   // the same network as SCL:
   "NTPserver".i_auxRetVal := RD_SYS_T(OUT => "NTPserver".dtl_Time, ENO => #_w1);
   IF #_w1 THEN
       "LSNTP_Server_DB"(init := "NTPserver".x_lEnable,   // "LSNTP_Server"
                         referenceId := "NTPserver".i_Reference,
                         lastTimeSet := "NTPserver".dtl_Time,
                         connID := 16#21,
                         hwID := "Local~Interfaccia_PROFINET_1");
   END_IF;
END_REGION
END_FUNCTION

FUNCTION "MV SKID (PE)" : Void   // FC45, LAD
TITLE = ModBus TCP for MVSKID Power Electronics
{ S7_Optimized_Access := 'TRUE' }
VERSION : 0.1
// stored: AutoNumber false, IsIECCheckEnabled false, SetENOAutomatically false, UDAEnableTagReadback false
   VAR_TEMP   // added for the SCL form of the ladder/FBD networks
      _w1 : Bool;
   END_VAR
BEGIN

REGION Network 1: Function Modbus Client
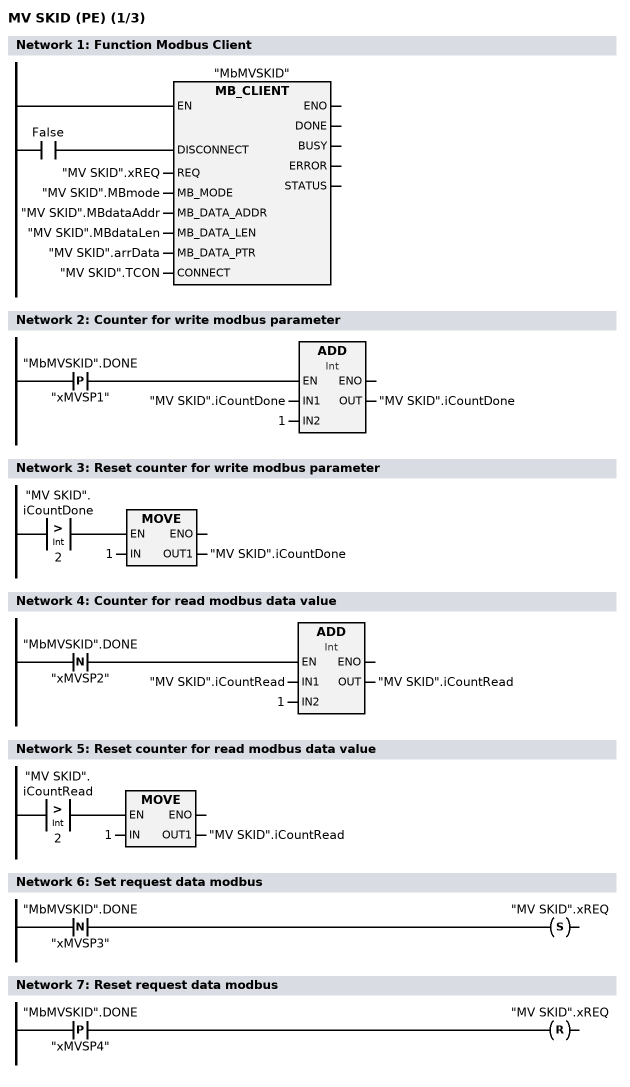
   RUNG wire#powerrail
      "MbMVSKID".MB_CLIENT(DISCONNECT := wire#w1, REQ := "MV SKID".xREQ, MB_MODE := "MV SKID".MBmode, MB_DATA_ADDR := "MV SKID".MBdataAddr, MB_DATA_LEN := "MV SKID".MBdataLen, MB_DATA_PTR := "MV SKID".arrData, CONNECT := "MV SKID".TCON, DONE =>, BUSY =>, ERROR =>, STATUS =>)
   END_RUNG
   RUNG wire#powerrail
      Contact( False )
   END_RUNG wire#w1
   // the same network as SCL:
   "MbMVSKID"(DISCONNECT := False,   // MB_CLIENT
              REQ := "MV SKID".xREQ,
              MB_MODE := "MV SKID".MBmode,
              MB_DATA_ADDR := "MV SKID".MBdataAddr,
              MB_DATA_LEN := "MV SKID".MBdataLen,
              MB_DATA_PTR := "MV SKID".arrData,
              CONNECT := "MV SKID".TCON);
END_REGION

REGION Network 2: Counter for write modbus parameter
   RUNG wire#powerrail
      P_Contact(operand := "MbMVSKID".DONE, bit := "xMVSP1")
      { S7_Templates := "SrcType := Int" } Add(in1 := "MV SKID".iCountDone, in2 := 1, out => "MV SKID".iCountDone)
   END_RUNG
   // the same network as SCL:
   #_w1 := "MbMVSKID".DONE AND NOT "xMVSP1";   // rising edge of "MbMVSKID".DONE
   "xMVSP1" := "MbMVSKID".DONE;
   IF #_w1 THEN "MV SKID".iCountDone := "MV SKID".iCountDone + 1; END_IF;
END_REGION

REGION Network 3: Reset counter for write modbus parameter
   RUNG wire#powerrail
      { S7_Templates := "SrcType := Int" } GT_Contact(in1 := "MV SKID".iCountDone, in2 := 2)
      Move(in := 1, out1 => "MV SKID".iCountDone)
   END_RUNG
   // the same network as SCL:
   IF "MV SKID".iCountDone > 2 THEN "MV SKID".iCountDone := 1; END_IF;
END_REGION

REGION Network 4: Counter for read modbus data value
   RUNG wire#powerrail
      N_Contact(operand := "MbMVSKID".DONE, bit := "xMVSP2")
      { S7_Templates := "SrcType := Int" } Add(in1 := "MV SKID".iCountRead, in2 := 1, out => "MV SKID".iCountRead)
   END_RUNG
   // the same network as SCL:
   #_w1 := NOT "MbMVSKID".DONE AND "xMVSP2";   // falling edge of "MbMVSKID".DONE
   "xMVSP2" := "MbMVSKID".DONE;
   IF #_w1 THEN "MV SKID".iCountRead := "MV SKID".iCountRead + 1; END_IF;
END_REGION

REGION Network 5: Reset counter for read modbus data value
   RUNG wire#powerrail
      { S7_Templates := "SrcType := Int" } GT_Contact(in1 := "MV SKID".iCountRead, in2 := 2)
      Move(in := 1, out1 => "MV SKID".iCountRead)
   END_RUNG
   // the same network as SCL:
   IF "MV SKID".iCountRead > 2 THEN "MV SKID".iCountRead := 1; END_IF;
END_REGION

REGION Network 6: Set request data modbus
   RUNG wire#powerrail
      N_Contact(operand := "MbMVSKID".DONE, bit := "xMVSP3")
      S_Coil( "MV SKID".xREQ )
   END_RUNG
   // the same network as SCL:
   #_w1 := NOT "MbMVSKID".DONE AND "xMVSP3";   // falling edge of "MbMVSKID".DONE
   "xMVSP3" := "MbMVSKID".DONE;
   IF #_w1 THEN "MV SKID".xREQ := TRUE; END_IF;
END_REGION

REGION Network 7: Reset request data modbus
   RUNG wire#powerrail
      P_Contact(operand := "MbMVSKID".DONE, bit := "xMVSP4")
      R_Coil( "MV SKID".xREQ )
   END_RUNG
   // the same network as SCL:
   #_w1 := "MbMVSKID".DONE AND NOT "xMVSP4";   // rising edge of "MbMVSKID".DONE
   "xMVSP4" := "MbMVSKID".DONE;
   IF #_w1 THEN "MV SKID".xREQ := FALSE; END_IF;
END_REGION

REGION Network 8: Write R_MVSKID parameter
